// TIA Portal V20 export
// export: Created 2025-12-01T14:57:01.3679822Z, ExportSetting None, DisplayName Totally Integrated Automation Portal, DisplayVersion V20 Update 3, DisplayName TIA Portal Openness, DisplayVersion V20 Update 3, DisplayName TIA Portal Version Control Interface, DisplayVersion V20 Update 3, DisplayName STEP 7 Professional, DisplayVersion V20 Update 3, DisplayName STEP 7 Safety, DisplayVersion V20 Update 2, DisplayName WinCC Basic/Comfort/Advanced, DisplayVersion V20 Update 3, DisplayName WinCC Professional, DisplayVersion V20 Update 3, DisplayName WinCC Unified, DisplayVersion V20 Update 3
FUNCTION "FC457_TL_TR_E1E3_S2_Aus" : Void   // FC457, LAD
{ S7_Optimized_Access := 'FALSE' }
AUTHOR : TLigero
NAME : 20180125
VERSION : 3.2
// FECHA:    27/07/2014  AUTOR: G.Martin
// INSTALACION: Magyar Posta
// //////////////////////////////////
// // Registro Incidencias   ////////
// //////////////////////////////////
// FECHA:21/10/14   AUTOR MODIFICACION: N.Rodriguez
// DESCRIPCION: 
// Adaptación de la función al estandar actual
// ULTIMA MODIFICACION: iñaki Arrondo por problemas detectados en la instalacion (ALKAR)
// stored: AutoNumber false, SetENOAutomatically false
   VAR_INPUT
      Mesa : UInt;
      En_Tension : Bool;
      pHsMx_E1 : Bool;
      pHsMx_E3 : Bool;
      pHsMx_S2 : Bool;
      TP_E1_UP : Bool;
      TP_E1_Dw : Bool;
      TP_E3_UP : Bool;
      TP_E3_Dw : Bool;
      Termico_E1_Tx : Bool;
      Termico_S2_Tx : Bool;
      Avance_E1_Tx_Ok : Bool;
      Avance_E3_Tx_Ok : Bool;   // será el retroceso de E1
      Avance_S2_Tx_Ok : Bool;
      PosTR_E1 : Bool;
      PosTR_S2 : Bool;
      AVTF_Ent_M1 : Bool;
      AVTF_Ent_M3 : Bool;
      NXT_Avance : Bool;
      PTF_Mx_MSig : Bool;
      V_CNT_ApHsMx_S2 : UDInt;   // Valor del Contador de ausencia en S2
      V_CNT_ApHsMx_E1 : UDInt;   // Valor del Contador de ausencia en E1
      V_CNT_ApHsMx_E3 : UDInt;   // Valor del Contador de ausencia en S3
      V_Paro : UDInt;
      V_TOut_Tx_Mx : UDInt;
      V_TOut_TR : UDInt;
      V_RepartoColector : UDInt;
   END_VAR
   VAR_OUTPUT
      PTF_Ent_M1 : Bool;
      PTF_Ent_M3 : Bool;
      AVTF_Mx_MSig : Bool;
   END_VAR
   VAR_IN_OUT
      Mem_tmp_Paro : Bool;
      MemAuxFN_E1 : Bool;
      MemFN_pHsE1 : Bool;
      MemFP_pHsE1 : Bool;
      MemAuxFN_E3 : Bool;
      MemFN_pHsE3 : Bool;
      MemAuxFN_S2 : Bool;
      MemFN_pHsS2 : Bool;
   END_VAR
   VAR_TEMP
      OK_Ausencia_Entrada : Bool;
      OK_Ausencia_salida : Bool;
      ok_vaciado : Bool;
      Error_Atasco : Bool;
      Error_TOut_TR : Bool;
      TEMP_MA_TR_PosE1E3 : Bool;
      TEMP_MA_TR_PosS2 : Bool;
      ok_tension : Bool;
      v_ausencia_entrada : UDInt;
   END_VAR
   VAR_TEMP   // added for the SCL form of the ladder/FBD networks
      _w1 : Bool;
      _w2 : Bool;
      _w3 : Bool;
      _w4 : Bool;
      _w5 : Bool;
      _w6 : Bool;
   END_VAR
BEGIN

REGION Network 1: Marca General Error
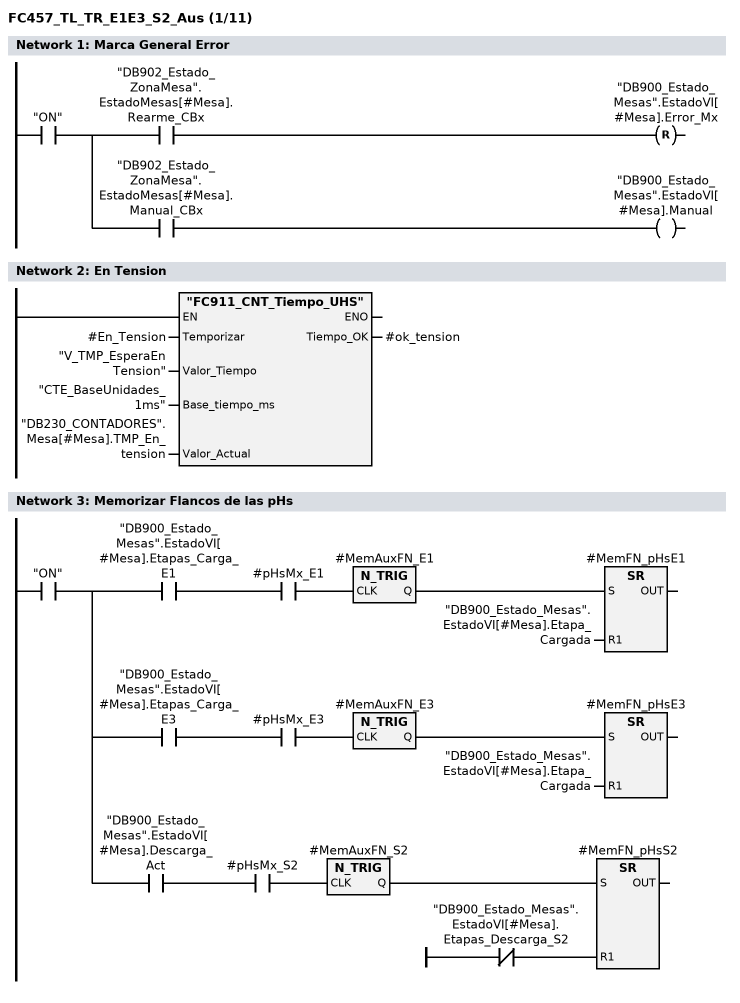
   RUNG wire#powerrail
      Contact( "ON" )
      wire#w1
      Contact( "DB902_Estado_ZonaMesa".EstadoMesas[#Mesa].Rearme_CBx )
      R_Coil( "DB900_Estado_Mesas".EstadoVI[#Mesa].Error_Mx )
   END_RUNG
   RUNG wire#w1
      Contact( "DB902_Estado_ZonaMesa".EstadoMesas[#Mesa].Manual_CBx )
      Coil( "DB900_Estado_Mesas".EstadoVI[#Mesa].Manual )
   END_RUNG
   // the same network as SCL:
   IF "ON" AND "DB902_Estado_ZonaMesa".EstadoMesas[#Mesa].Rearme_CBx THEN
       "DB900_Estado_Mesas".EstadoVI[#Mesa].Error_Mx := FALSE;
   END_IF;
   "DB900_Estado_Mesas".EstadoVI[#Mesa].Manual := "ON" AND "DB902_Estado_ZonaMesa".EstadoMesas[#Mesa].Manual_CBx;
END_REGION

REGION Network 2: En Tension
   RUNG wire#powerrail
      "FC911_CNT_Tiempo_UHS"(Temporizar := #En_Tension, Valor_Tiempo := "V_TMP_EsperaEnTension", Base_tiempo_ms := "CTE_BaseUnidades_1ms", Valor_Actual := "DB230_CONTADORES".Mesa[#Mesa].TMP_En_tension, Tiempo_OK => #ok_tension)
   END_RUNG
   // the same network as SCL:
   "FC911_CNT_Tiempo_UHS"(Temporizar := #En_Tension,
                          Valor_Tiempo := "V_TMP_EsperaEnTension",
                          Base_tiempo_ms := "CTE_BaseUnidades_1ms",
                          Valor_Actual := "DB230_CONTADORES".Mesa[#Mesa].TMP_En_tension,
                          Tiempo_OK => #ok_tension);
END_REGION

REGION Network 3: Memorizar Flancos de las pHs
   RUNG wire#powerrail
      Contact( "ON" )
      wire#w1
      Contact( "DB900_Estado_Mesas".EstadoVI[#Mesa].Etapas_Carga_E1 )
      Contact( #pHsMx_E1 )
      N_Trig( #MemAuxFN_E1 )
      S_SR(operand := #MemFN_pHsE1, r1 := "DB900_Estado_Mesas".EstadoVI[#Mesa].Etapa_Cargada)
   END_RUNG
   RUNG wire#w1
      Contact( "DB900_Estado_Mesas".EstadoVI[#Mesa].Etapas_Carga_E3 )
      Contact( #pHsMx_E3 )
      N_Trig( #MemAuxFN_E3 )
      S_SR(operand := #MemFN_pHsE3, r1 := "DB900_Estado_Mesas".EstadoVI[#Mesa].Etapa_Cargada)
   END_RUNG
   RUNG wire#w1
      Contact( "DB900_Estado_Mesas".EstadoVI[#Mesa].Descarga_Act )
      Contact( #pHsMx_S2 )
      N_Trig( #MemAuxFN_S2 )
      S_SR(operand := #MemFN_pHsS2, r1 := wire#w2)
   END_RUNG
   RUNG wire#powerrail
      I_Contact( "DB900_Estado_Mesas".EstadoVI[#Mesa].Etapas_Descarga_S2 )
   END_RUNG wire#w2
   // the same network as SCL:
   #_w1 := "ON" AND "DB900_Estado_Mesas".EstadoVI[#Mesa].Etapas_Carga_E1 AND #pHsMx_E1;
   #_w2 := NOT #_w1 AND #MemAuxFN_E1;   // falling edge
   #MemAuxFN_E1 := #_w1;
   IF #_w2 THEN
       #MemFN_pHsE1 := TRUE;   // SR flip-flop
   END_IF;
   IF "DB900_Estado_Mesas".EstadoVI[#Mesa].Etapa_Cargada THEN #MemFN_pHsE1 := FALSE; END_IF;
   #_w3 := "ON" AND "DB900_Estado_Mesas".EstadoVI[#Mesa].Etapas_Carga_E3 AND #pHsMx_E3;
   #_w4 := NOT #_w3 AND #MemAuxFN_E3;   // falling edge
   #MemAuxFN_E3 := #_w3;
   IF #_w4 THEN
       #MemFN_pHsE3 := TRUE;   // SR flip-flop
   END_IF;
   IF "DB900_Estado_Mesas".EstadoVI[#Mesa].Etapa_Cargada THEN #MemFN_pHsE3 := FALSE; END_IF;
   #_w5 := "ON" AND "DB900_Estado_Mesas".EstadoVI[#Mesa].Descarga_Act AND #pHsMx_S2;
   #_w6 := NOT #_w5 AND #MemAuxFN_S2;   // falling edge
   #MemAuxFN_S2 := #_w5;
   IF #_w6 THEN
       #MemFN_pHsS2 := TRUE;   // SR flip-flop
   END_IF;
   IF NOT "DB900_Estado_Mesas".EstadoVI[#Mesa].Etapas_Descarga_S2 THEN #MemFN_pHsS2 := FALSE; END_IF;
END_REGION

REGION Network 4: contador vaciado
   // Contador ausencia
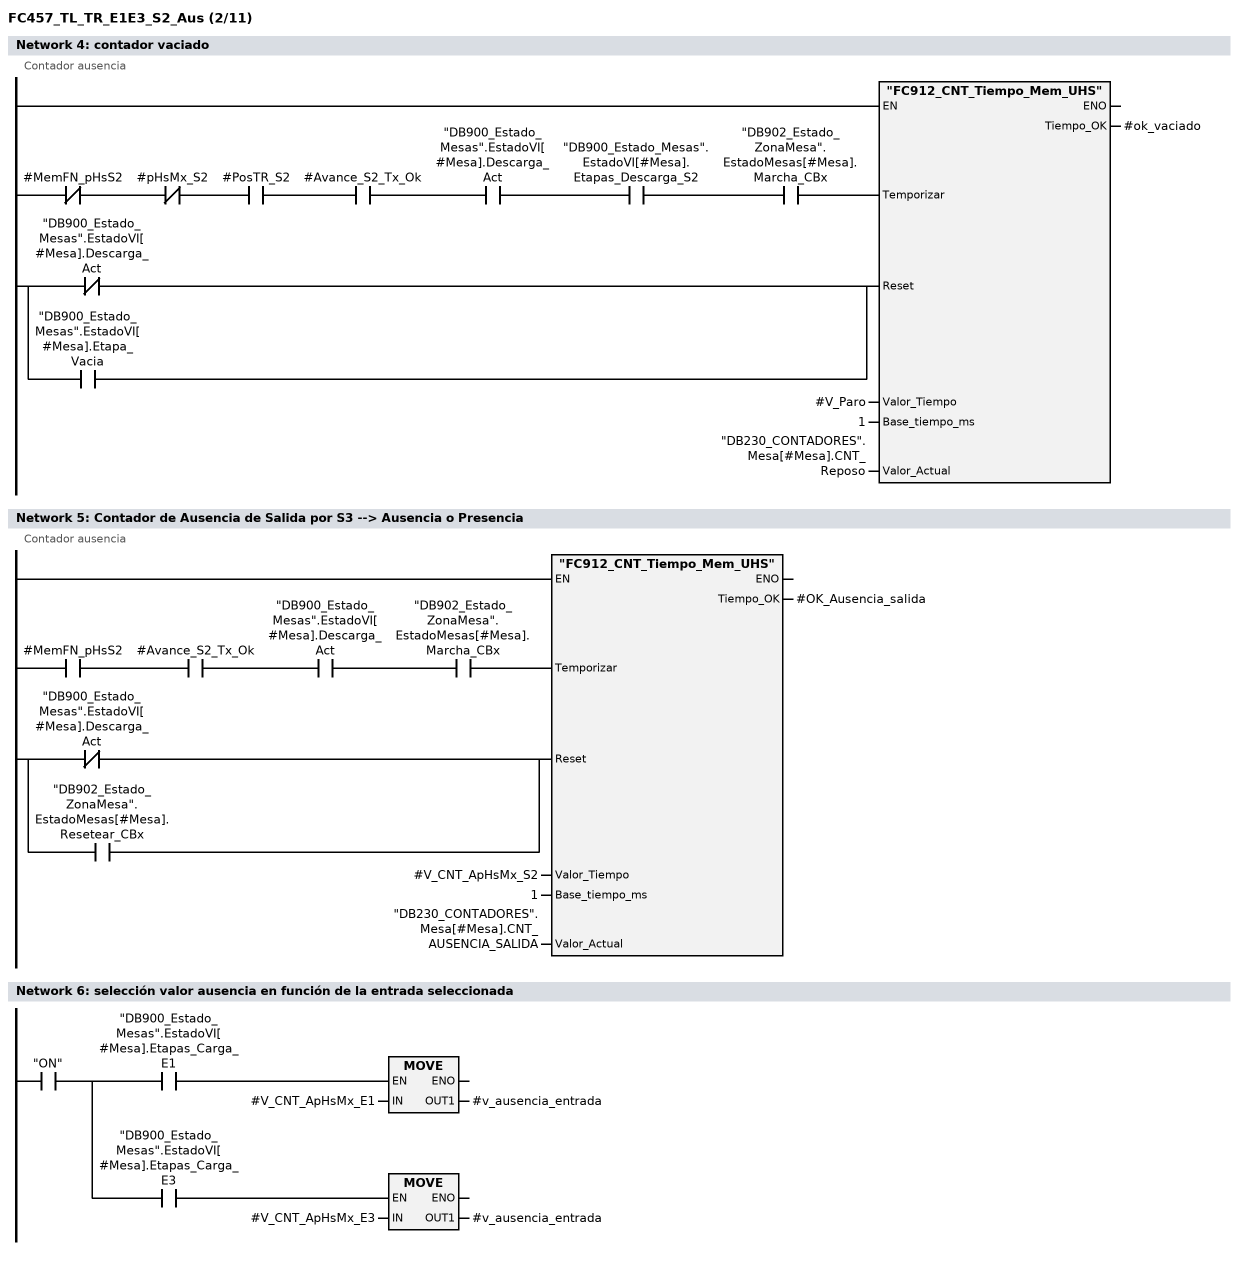
   RUNG wire#powerrail
      "FC912_CNT_Tiempo_Mem_UHS"(Temporizar := wire#w1, Reset := wire#w2, Valor_Tiempo := #V_Paro, Base_tiempo_ms := 1, Valor_Actual := "DB230_CONTADORES".Mesa[#Mesa].CNT_Reposo, Tiempo_OK => #ok_vaciado)
   END_RUNG
   RUNG wire#powerrail
      I_Contact( #MemFN_pHsS2 )
      I_Contact( #pHsMx_S2 )
      Contact( #PosTR_S2 )
      Contact( #Avance_S2_Tx_Ok )
      Contact( "DB900_Estado_Mesas".EstadoVI[#Mesa].Descarga_Act )
      Contact( "DB900_Estado_Mesas".EstadoVI[#Mesa].Etapas_Descarga_S2 )
      Contact( "DB902_Estado_ZonaMesa".EstadoMesas[#Mesa].Marcha_CBx )
   END_RUNG wire#w1
   RUNG wire#powerrail
      I_Contact( "DB900_Estado_Mesas".EstadoVI[#Mesa].Descarga_Act )
   END_RUNG wire#w2
   RUNG wire#powerrail
      Contact( "DB900_Estado_Mesas".EstadoVI[#Mesa].Etapa_Vacia )
   END_RUNG wire#w2
   // the same network as SCL:
   "FC912_CNT_Tiempo_Mem_UHS"(Temporizar := NOT #MemFN_pHsS2 AND NOT #pHsMx_S2 AND #PosTR_S2 AND #Avance_S2_Tx_Ok AND "DB900_Estado_Mesas".EstadoVI[#Mesa].Descarga_Act AND "DB900_Estado_Mesas".EstadoVI[#Mesa].Etapas_Descarga_S2 AND "DB902_Estado_ZonaMesa".EstadoMesas[#Mesa].Marcha_CBx,
                           Reset := NOT "DB900_Estado_Mesas".EstadoVI[#Mesa].Descarga_Act OR "DB900_Estado_Mesas".EstadoVI[#Mesa].Etapa_Vacia,
                           Valor_Tiempo := #V_Paro,
                           Base_tiempo_ms := 1,
                           Valor_Actual := "DB230_CONTADORES".Mesa[#Mesa].CNT_Reposo,
                           Tiempo_OK => #ok_vaciado);
END_REGION

REGION Network 5: Contador de Ausencia de Salida por S3 --> Ausencia o Presencia
   // Contador ausencia
   RUNG wire#powerrail
      "FC912_CNT_Tiempo_Mem_UHS"(Temporizar := wire#w1, Reset := wire#w2, Valor_Tiempo := #V_CNT_ApHsMx_S2, Base_tiempo_ms := 1, Valor_Actual := "DB230_CONTADORES".Mesa[#Mesa].CNT_AUSENCIA_SALIDA, Tiempo_OK => #OK_Ausencia_salida)
   END_RUNG
   RUNG wire#powerrail
      Contact( #MemFN_pHsS2 )
      Contact( #Avance_S2_Tx_Ok )
      Contact( "DB900_Estado_Mesas".EstadoVI[#Mesa].Descarga_Act )
      Contact( "DB902_Estado_ZonaMesa".EstadoMesas[#Mesa].Marcha_CBx )
   END_RUNG wire#w1
   RUNG wire#powerrail
      I_Contact( "DB900_Estado_Mesas".EstadoVI[#Mesa].Descarga_Act )
   END_RUNG wire#w2
   RUNG wire#powerrail
      Contact( "DB902_Estado_ZonaMesa".EstadoMesas[#Mesa].Resetear_CBx )
   END_RUNG wire#w2
   // the same network as SCL:
   "FC912_CNT_Tiempo_Mem_UHS"(Temporizar := #MemFN_pHsS2 AND #Avance_S2_Tx_Ok AND "DB900_Estado_Mesas".EstadoVI[#Mesa].Descarga_Act AND "DB902_Estado_ZonaMesa".EstadoMesas[#Mesa].Marcha_CBx,
                           Reset := NOT "DB900_Estado_Mesas".EstadoVI[#Mesa].Descarga_Act OR "DB902_Estado_ZonaMesa".EstadoMesas[#Mesa].Resetear_CBx,
                           Valor_Tiempo := #V_CNT_ApHsMx_S2,
                           Base_tiempo_ms := 1,
                           Valor_Actual := "DB230_CONTADORES".Mesa[#Mesa].CNT_AUSENCIA_SALIDA,
                           Tiempo_OK => #OK_Ausencia_salida);
END_REGION

REGION Network 6: selección valor ausencia en función de la entrada seleccionada
   RUNG wire#powerrail
      Contact( "ON" )
      wire#w1
      Contact( "DB900_Estado_Mesas".EstadoVI[#Mesa].Etapas_Carga_E1 )
      Move(in := #V_CNT_ApHsMx_E1, out1 => #v_ausencia_entrada)
   END_RUNG
   RUNG wire#w1
      Contact( "DB900_Estado_Mesas".EstadoVI[#Mesa].Etapas_Carga_E3 )
      Move(in := #V_CNT_ApHsMx_E3, out1 => #v_ausencia_entrada)
   END_RUNG
   // the same network as SCL:
   IF "ON" AND "DB900_Estado_Mesas".EstadoVI[#Mesa].Etapas_Carga_E1 THEN
       #v_ausencia_entrada := #V_CNT_ApHsMx_E1;
   END_IF;
   IF "ON" AND "DB900_Estado_Mesas".EstadoVI[#Mesa].Etapas_Carga_E3 THEN
       #v_ausencia_entrada := #V_CNT_ApHsMx_E3;
   END_IF;
END_REGION

REGION Network 7: Contador de Ausencia de Entrada
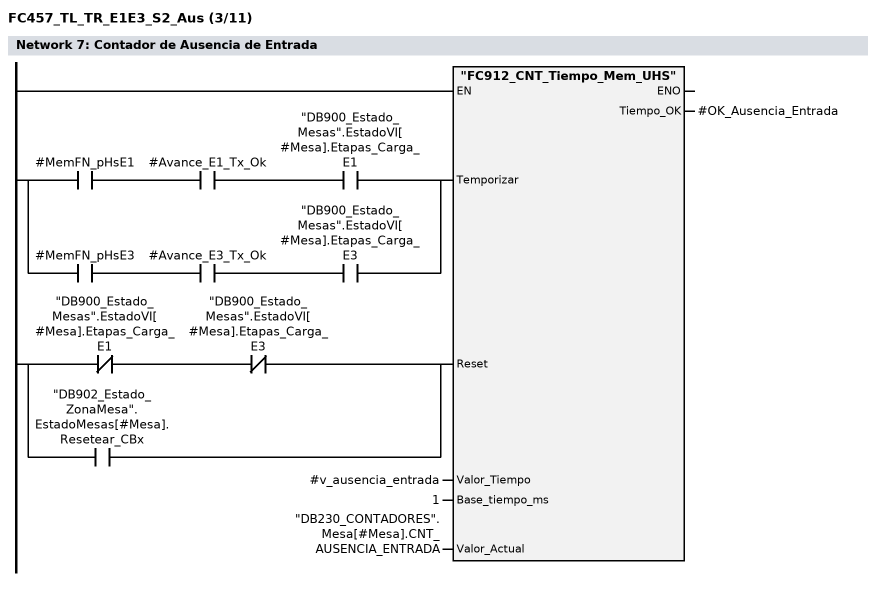
   RUNG wire#powerrail
      "FC912_CNT_Tiempo_Mem_UHS"(Temporizar := wire#w1, Reset := wire#w2, Valor_Tiempo := #v_ausencia_entrada, Base_tiempo_ms := 1, Valor_Actual := "DB230_CONTADORES".Mesa[#Mesa].CNT_AUSENCIA_ENTRADA, Tiempo_OK => #OK_Ausencia_Entrada)
   END_RUNG
   RUNG wire#powerrail
      Contact( #MemFN_pHsE1 )
      Contact( #Avance_E1_Tx_Ok )
      Contact( "DB900_Estado_Mesas".EstadoVI[#Mesa].Etapas_Carga_E1 )
   END_RUNG wire#w1
   RUNG wire#powerrail
      Contact( #MemFN_pHsE3 )
      Contact( #Avance_E3_Tx_Ok )
      Contact( "DB900_Estado_Mesas".EstadoVI[#Mesa].Etapas_Carga_E3 )
   END_RUNG wire#w1
   RUNG wire#powerrail
      I_Contact( "DB900_Estado_Mesas".EstadoVI[#Mesa].Etapas_Carga_E1 )
      I_Contact( "DB900_Estado_Mesas".EstadoVI[#Mesa].Etapas_Carga_E3 )
   END_RUNG wire#w2
   RUNG wire#powerrail
      Contact( "DB902_Estado_ZonaMesa".EstadoMesas[#Mesa].Resetear_CBx )
   END_RUNG wire#w2
   // the same network as SCL:
   "FC912_CNT_Tiempo_Mem_UHS"(Temporizar := (#MemFN_pHsE1 AND #Avance_E1_Tx_Ok AND "DB900_Estado_Mesas".EstadoVI[#Mesa].Etapas_Carga_E1) OR (#MemFN_pHsE3 AND #Avance_E3_Tx_Ok AND "DB900_Estado_Mesas".EstadoVI[#Mesa].Etapas_Carga_E3),
                           Reset := (NOT "DB900_Estado_Mesas".EstadoVI[#Mesa].Etapas_Carga_E1 AND NOT "DB900_Estado_Mesas".EstadoVI[#Mesa].Etapas_Carga_E3) OR "DB902_Estado_ZonaMesa".EstadoMesas[#Mesa].Resetear_CBx,
                           Valor_Tiempo := #v_ausencia_entrada,
                           Base_tiempo_ms := 1,
                           Valor_Actual := "DB230_CONTADORES".Mesa[#Mesa].CNT_AUSENCIA_ENTRADA,
                           Tiempo_OK => #OK_Ausencia_Entrada);
END_REGION

REGION Network 8: Temporizador de PARO
   // Modif Dani: El contador se activa además de con MA_avance_Tx, con el 
   // MA_Avance_TR, pq sino, no se resetean las variables de Mem_Act_E1, E2 tras un 
   // reset
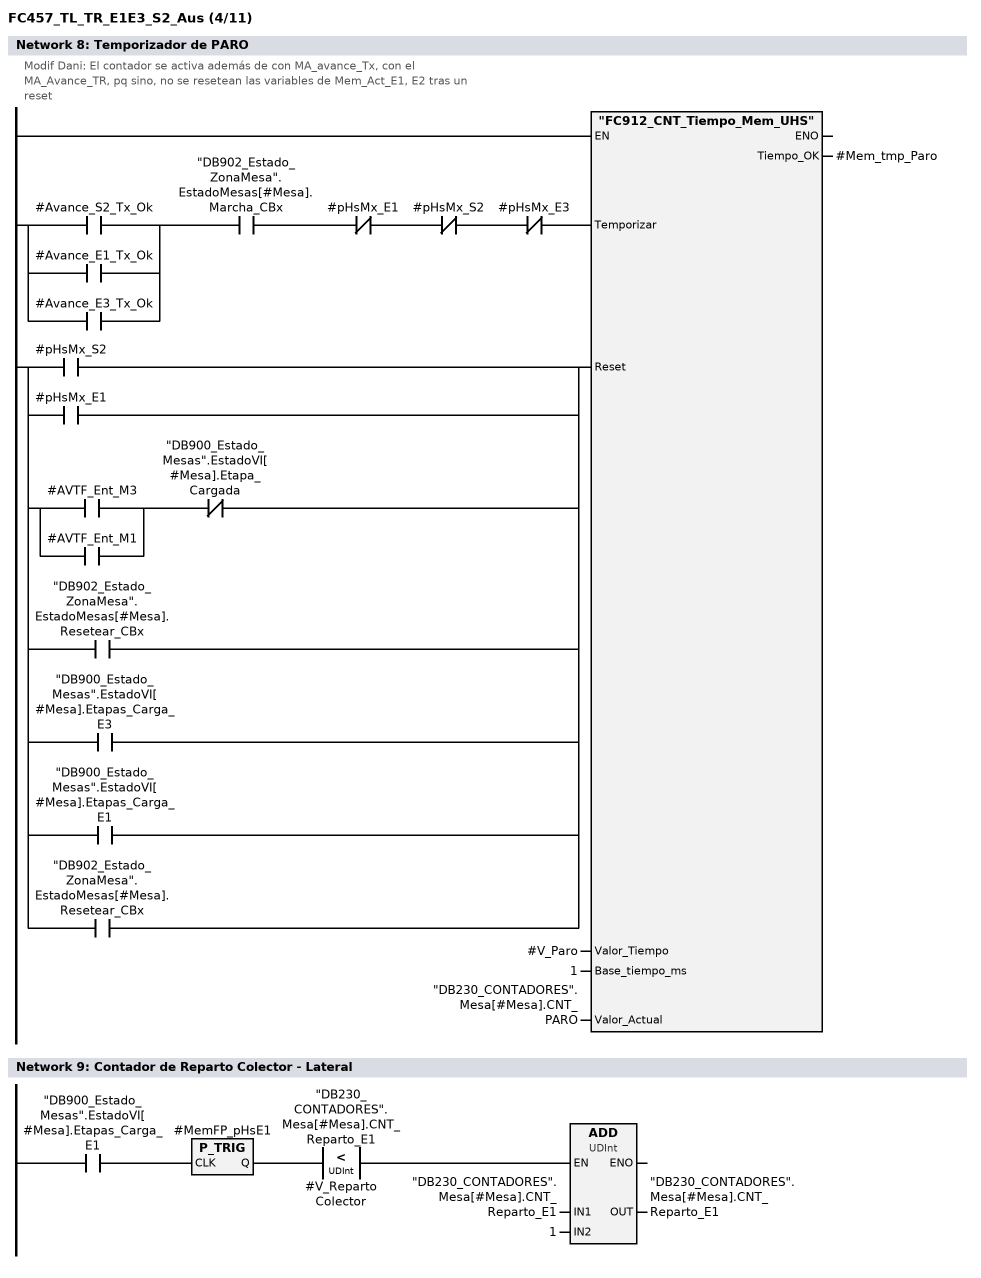
   RUNG wire#powerrail
      "FC912_CNT_Tiempo_Mem_UHS"(Temporizar := wire#w2, Reset := wire#w4, Valor_Tiempo := #V_Paro, Base_tiempo_ms := 1, Valor_Actual := "DB230_CONTADORES".Mesa[#Mesa].CNT_PARO, Tiempo_OK => #Mem_tmp_Paro)
   END_RUNG
   RUNG wire#powerrail
      Contact( #Avance_S2_Tx_Ok )
      wire#w1
      Contact( "DB902_Estado_ZonaMesa".EstadoMesas[#Mesa].Marcha_CBx )
      I_Contact( #pHsMx_E1 )
      I_Contact( #pHsMx_S2 )
      I_Contact( #pHsMx_E3 )
   END_RUNG wire#w2
   RUNG wire#powerrail
      Contact( #Avance_E1_Tx_Ok )
   END_RUNG wire#w1
   RUNG wire#powerrail
      Contact( #Avance_E3_Tx_Ok )
   END_RUNG wire#w1
   RUNG wire#powerrail
      Contact( #pHsMx_S2 )
   END_RUNG wire#w4
   RUNG wire#powerrail
      Contact( #pHsMx_E1 )
   END_RUNG wire#w4
   RUNG wire#powerrail
      Contact( #AVTF_Ent_M3 )
      wire#w3
      I_Contact( "DB900_Estado_Mesas".EstadoVI[#Mesa].Etapa_Cargada )
   END_RUNG wire#w4
   RUNG wire#powerrail
      Contact( #AVTF_Ent_M1 )
   END_RUNG wire#w3
   RUNG wire#powerrail
      Contact( "DB902_Estado_ZonaMesa".EstadoMesas[#Mesa].Resetear_CBx )
   END_RUNG wire#w4
   RUNG wire#powerrail
      Contact( "DB900_Estado_Mesas".EstadoVI[#Mesa].Etapas_Carga_E3 )
   END_RUNG wire#w4
   RUNG wire#powerrail
      Contact( "DB900_Estado_Mesas".EstadoVI[#Mesa].Etapas_Carga_E1 )
   END_RUNG wire#w4
   RUNG wire#powerrail
      Contact( "DB902_Estado_ZonaMesa".EstadoMesas[#Mesa].Resetear_CBx )
   END_RUNG wire#w4
   // the same network as SCL:
   "FC912_CNT_Tiempo_Mem_UHS"(Temporizar := (#Avance_S2_Tx_Ok OR #Avance_E1_Tx_Ok OR #Avance_E3_Tx_Ok) AND "DB902_Estado_ZonaMesa".EstadoMesas[#Mesa].Marcha_CBx AND NOT #pHsMx_E1 AND NOT #pHsMx_S2 AND NOT #pHsMx_E3,
                           Reset := #pHsMx_S2 OR #pHsMx_E1 OR ((#AVTF_Ent_M3 OR #AVTF_Ent_M1) AND NOT "DB900_Estado_Mesas".EstadoVI[#Mesa].Etapa_Cargada) OR "DB902_Estado_ZonaMesa".EstadoMesas[#Mesa].Resetear_CBx OR "DB900_Estado_Mesas".EstadoVI[#Mesa].Etapas_Carga_E3 OR "DB900_Estado_Mesas".EstadoVI[#Mesa].Etapas_Carga_E1 OR "DB902_Estado_ZonaMesa".EstadoMesas[#Mesa].Resetear_CBx,
                           Valor_Tiempo := #V_Paro,
                           Base_tiempo_ms := 1,
                           Valor_Actual := "DB230_CONTADORES".Mesa[#Mesa].CNT_PARO,
                           Tiempo_OK => #Mem_tmp_Paro);
END_REGION

REGION Network 9: Contador de Reparto Colector - Lateral
   RUNG wire#powerrail
      Contact( "DB900_Estado_Mesas".EstadoVI[#Mesa].Etapas_Carga_E1 )
      P_Trig( #MemFP_pHsE1 )
      { S7_Templates := "SrcType := UDInt" } LT_Contact(in1 := "DB230_CONTADORES".Mesa[#Mesa].CNT_Reparto_E1, in2 := #V_RepartoColector)
      { S7_Templates := "SrcType := UDInt"; S7_GenerateENO := "TRUE" } Add(in1 := "DB230_CONTADORES".Mesa[#Mesa].CNT_Reparto_E1, in2 := 1, out => "DB230_CONTADORES".Mesa[#Mesa].CNT_Reparto_E1)
   END_RUNG
   // the same network as SCL:
   #_w1 := "DB900_Estado_Mesas".EstadoVI[#Mesa].Etapas_Carga_E1 AND NOT #MemFP_pHsE1;   // rising edge
   #MemFP_pHsE1 := "DB900_Estado_Mesas".EstadoVI[#Mesa].Etapas_Carga_E1;
   IF #_w1 AND ("DB230_CONTADORES".Mesa[#Mesa].CNT_Reparto_E1 < #V_RepartoColector) THEN
       "DB230_CONTADORES".Mesa[#Mesa].CNT_Reparto_E1 := "DB230_CONTADORES".Mesa[#Mesa].CNT_Reparto_E1 + 1;
   END_IF;
END_REGION

REGION Network 10
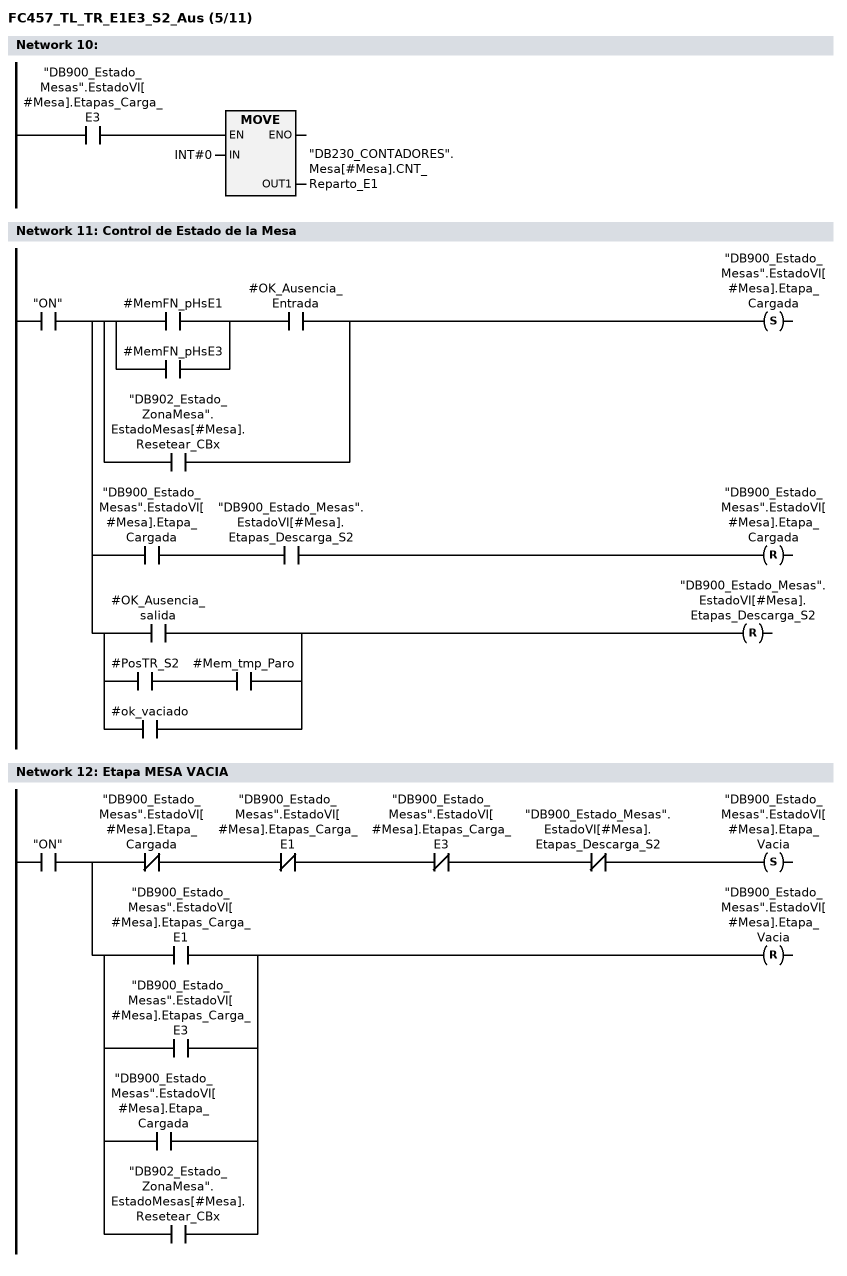
   RUNG wire#powerrail
      Contact( "DB900_Estado_Mesas".EstadoVI[#Mesa].Etapas_Carga_E3 )
      { S7_GenerateENO := "TRUE" } Move(in := INT#0, out1 => "DB230_CONTADORES".Mesa[#Mesa].CNT_Reparto_E1)
   END_RUNG
   // the same network as SCL:
   IF "DB900_Estado_Mesas".EstadoVI[#Mesa].Etapas_Carga_E3 THEN
       "DB230_CONTADORES".Mesa[#Mesa].CNT_Reparto_E1 := INT#0;
   END_IF;
END_REGION

REGION Network 11: Control de Estado de la Mesa
   RUNG wire#powerrail
      Contact( "ON" )
      wire#w1
      Contact( #MemFN_pHsE1 )
      wire#w2
      Contact( #OK_Ausencia_Entrada )
      wire#w3
      S_Coil( "DB900_Estado_Mesas".EstadoVI[#Mesa].Etapa_Cargada )
   END_RUNG
   RUNG wire#w1
      Contact( #MemFN_pHsE3 )
   END_RUNG wire#w2
   RUNG wire#w1
      Contact( "DB902_Estado_ZonaMesa".EstadoMesas[#Mesa].Resetear_CBx )
   END_RUNG wire#w3
   RUNG wire#w1
      Contact( "DB900_Estado_Mesas".EstadoVI[#Mesa].Etapa_Cargada )
      Contact( "DB900_Estado_Mesas".EstadoVI[#Mesa].Etapas_Descarga_S2 )
      R_Coil( "DB900_Estado_Mesas".EstadoVI[#Mesa].Etapa_Cargada )
   END_RUNG
   RUNG wire#w1
      Contact( #OK_Ausencia_salida )
      wire#w4
      R_Coil( "DB900_Estado_Mesas".EstadoVI[#Mesa].Etapas_Descarga_S2 )
   END_RUNG
   RUNG wire#w1
      Contact( #PosTR_S2 )
      Contact( #Mem_tmp_Paro )
   END_RUNG wire#w4
   RUNG wire#w1
      Contact( #ok_vaciado )
   END_RUNG wire#w4
   // the same network as SCL:
   IF "ON" AND (((#MemFN_pHsE1 OR #MemFN_pHsE3) AND #OK_Ausencia_Entrada) OR "DB902_Estado_ZonaMesa".EstadoMesas[#Mesa].Resetear_CBx) THEN
       "DB900_Estado_Mesas".EstadoVI[#Mesa].Etapa_Cargada := TRUE;
   END_IF;
   IF "ON" AND "DB900_Estado_Mesas".EstadoVI[#Mesa].Etapa_Cargada AND "DB900_Estado_Mesas".EstadoVI[#Mesa].Etapas_Descarga_S2 THEN
       "DB900_Estado_Mesas".EstadoVI[#Mesa].Etapa_Cargada := FALSE;
   END_IF;
   IF "ON" AND (#OK_Ausencia_salida OR (#PosTR_S2 AND #Mem_tmp_Paro) OR #ok_vaciado) THEN
       "DB900_Estado_Mesas".EstadoVI[#Mesa].Etapas_Descarga_S2 := FALSE;
   END_IF;
END_REGION

REGION Network 12: Etapa MESA VACIA
   RUNG wire#powerrail
      Contact( "ON" )
      wire#w1
      I_Contact( "DB900_Estado_Mesas".EstadoVI[#Mesa].Etapa_Cargada )
      I_Contact( "DB900_Estado_Mesas".EstadoVI[#Mesa].Etapas_Carga_E1 )
      I_Contact( "DB900_Estado_Mesas".EstadoVI[#Mesa].Etapas_Carga_E3 )
      I_Contact( "DB900_Estado_Mesas".EstadoVI[#Mesa].Etapas_Descarga_S2 )
      S_Coil( "DB900_Estado_Mesas".EstadoVI[#Mesa].Etapa_Vacia )
   END_RUNG
   RUNG wire#w1
      Contact( "DB900_Estado_Mesas".EstadoVI[#Mesa].Etapas_Carga_E1 )
      wire#w2
      R_Coil( "DB900_Estado_Mesas".EstadoVI[#Mesa].Etapa_Vacia )
   END_RUNG
   RUNG wire#w1
      Contact( "DB900_Estado_Mesas".EstadoVI[#Mesa].Etapas_Carga_E3 )
   END_RUNG wire#w2
   RUNG wire#w1
      Contact( "DB900_Estado_Mesas".EstadoVI[#Mesa].Etapa_Cargada )
   END_RUNG wire#w2
   RUNG wire#w1
      Contact( "DB902_Estado_ZonaMesa".EstadoMesas[#Mesa].Resetear_CBx )
   END_RUNG wire#w2
   // the same network as SCL:
   IF "ON" AND NOT "DB900_Estado_Mesas".EstadoVI[#Mesa].Etapa_Cargada AND NOT "DB900_Estado_Mesas".EstadoVI[#Mesa].Etapas_Carga_E1 AND NOT "DB900_Estado_Mesas".EstadoVI[#Mesa].Etapas_Carga_E3 AND NOT "DB900_Estado_Mesas".EstadoVI[#Mesa].Etapas_Descarga_S2 THEN
       "DB900_Estado_Mesas".EstadoVI[#Mesa].Etapa_Vacia := TRUE;
   END_IF;
   IF "ON" AND ("DB900_Estado_Mesas".EstadoVI[#Mesa].Etapas_Carga_E1 OR "DB900_Estado_Mesas".EstadoVI[#Mesa].Etapas_Carga_E3 OR "DB900_Estado_Mesas".EstadoVI[#Mesa].Etapa_Cargada OR "DB902_Estado_ZonaMesa".EstadoMesas[#Mesa].Resetear_CBx) THEN
       "DB900_Estado_Mesas".EstadoVI[#Mesa].Etapa_Vacia := FALSE;
   END_IF;
END_REGION

REGION Network 13
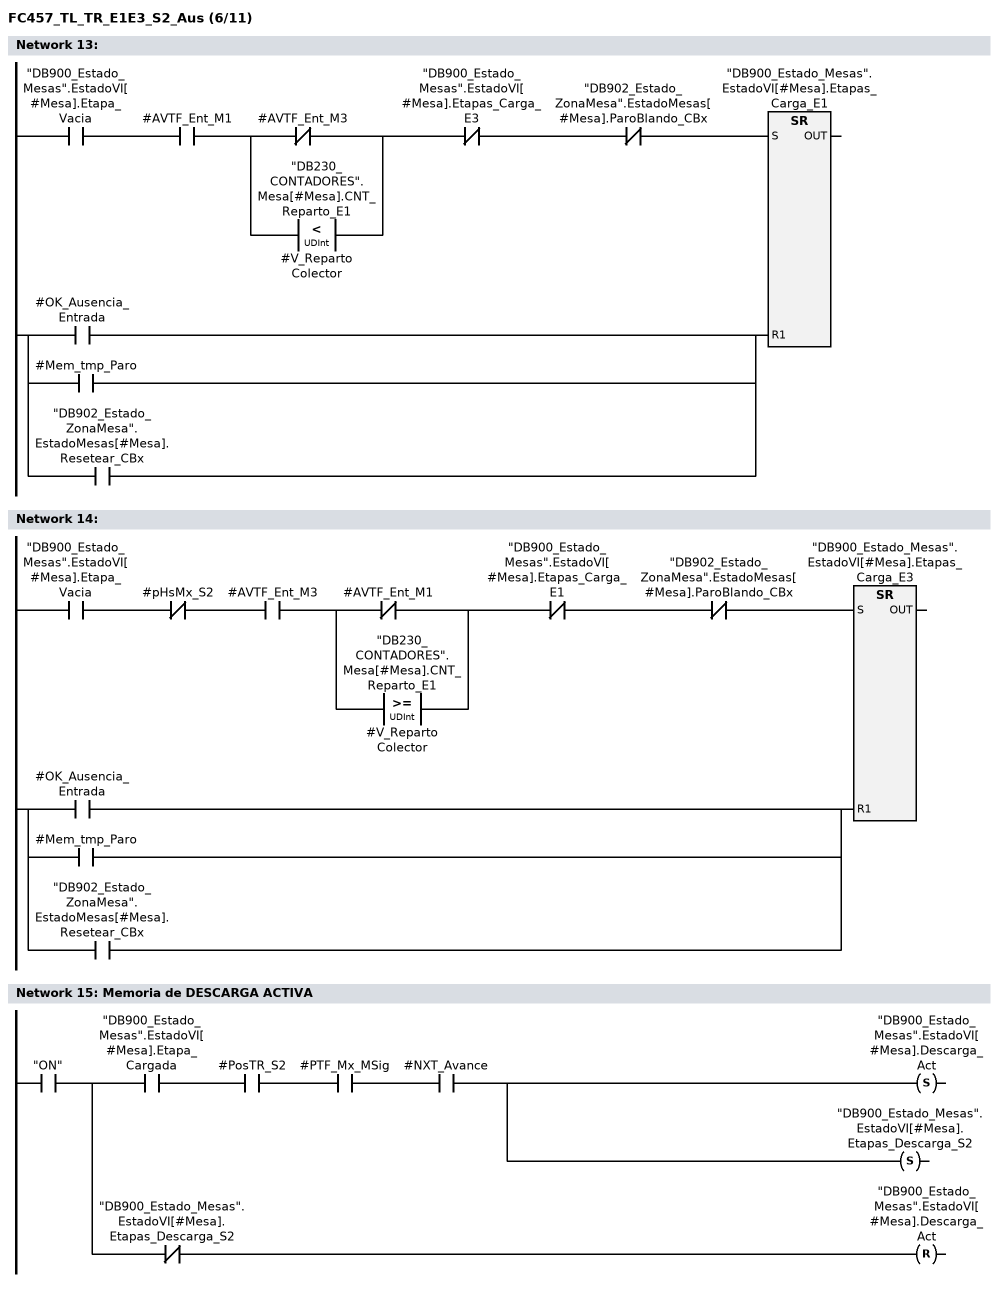
   RUNG wire#powerrail
      Contact( "DB900_Estado_Mesas".EstadoVI[#Mesa].Etapa_Vacia )
      Contact( #AVTF_Ent_M1 )
      wire#w1
      I_Contact( #AVTF_Ent_M3 )
      wire#w2
      I_Contact( "DB900_Estado_Mesas".EstadoVI[#Mesa].Etapas_Carga_E3 )
      I_Contact( "DB902_Estado_ZonaMesa".EstadoMesas[#Mesa].ParoBlando_CBx )
      S_SR(operand := "DB900_Estado_Mesas".EstadoVI[#Mesa].Etapas_Carga_E1, r1 := wire#w3)
   END_RUNG
   RUNG wire#w1
      { S7_Templates := "SrcType := UDInt" } LT_Contact(in1 := "DB230_CONTADORES".Mesa[#Mesa].CNT_Reparto_E1, in2 := #V_RepartoColector)
   END_RUNG wire#w2
   RUNG wire#powerrail
      Contact( #OK_Ausencia_Entrada )
   END_RUNG wire#w3
   RUNG wire#powerrail
      Contact( #Mem_tmp_Paro )
   END_RUNG wire#w3
   RUNG wire#powerrail
      Contact( "DB902_Estado_ZonaMesa".EstadoMesas[#Mesa].Resetear_CBx )
   END_RUNG wire#w3
   // the same network as SCL:
   #_w1 := #OK_Ausencia_Entrada OR #Mem_tmp_Paro OR "DB902_Estado_ZonaMesa".EstadoMesas[#Mesa].Resetear_CBx;
   IF "DB900_Estado_Mesas".EstadoVI[#Mesa].Etapa_Vacia AND #AVTF_Ent_M1 AND (NOT #AVTF_Ent_M3 OR ("DB230_CONTADORES".Mesa[#Mesa].CNT_Reparto_E1 < #V_RepartoColector)) AND NOT "DB900_Estado_Mesas".EstadoVI[#Mesa].Etapas_Carga_E3 AND NOT "DB902_Estado_ZonaMesa".EstadoMesas[#Mesa].ParoBlando_CBx THEN
       "DB900_Estado_Mesas".EstadoVI[#Mesa].Etapas_Carga_E1 := TRUE;   // SR flip-flop
   END_IF;
   IF #_w1 THEN "DB900_Estado_Mesas".EstadoVI[#Mesa].Etapas_Carga_E1 := FALSE; END_IF;
END_REGION

REGION Network 14
   RUNG wire#powerrail
      Contact( "DB900_Estado_Mesas".EstadoVI[#Mesa].Etapa_Vacia )
      I_Contact( #pHsMx_S2 )
      Contact( #AVTF_Ent_M3 )
      wire#w1
      I_Contact( #AVTF_Ent_M1 )
      wire#w2
      I_Contact( "DB900_Estado_Mesas".EstadoVI[#Mesa].Etapas_Carga_E1 )
      I_Contact( "DB902_Estado_ZonaMesa".EstadoMesas[#Mesa].ParoBlando_CBx )
      S_SR(operand := "DB900_Estado_Mesas".EstadoVI[#Mesa].Etapas_Carga_E3, r1 := wire#w3)
   END_RUNG
   RUNG wire#w1
      { S7_Templates := "SrcType := UDInt" } GE_Contact(in1 := "DB230_CONTADORES".Mesa[#Mesa].CNT_Reparto_E1, in2 := #V_RepartoColector)
   END_RUNG wire#w2
   RUNG wire#powerrail
      Contact( #OK_Ausencia_Entrada )
   END_RUNG wire#w3
   RUNG wire#powerrail
      Contact( #Mem_tmp_Paro )
   END_RUNG wire#w3
   RUNG wire#powerrail
      Contact( "DB902_Estado_ZonaMesa".EstadoMesas[#Mesa].Resetear_CBx )
   END_RUNG wire#w3
   // the same network as SCL:
   #_w1 := #OK_Ausencia_Entrada OR #Mem_tmp_Paro OR "DB902_Estado_ZonaMesa".EstadoMesas[#Mesa].Resetear_CBx;
   IF "DB900_Estado_Mesas".EstadoVI[#Mesa].Etapa_Vacia AND NOT #pHsMx_S2 AND #AVTF_Ent_M3 AND (NOT #AVTF_Ent_M1 OR ("DB230_CONTADORES".Mesa[#Mesa].CNT_Reparto_E1 >= #V_RepartoColector)) AND NOT "DB900_Estado_Mesas".EstadoVI[#Mesa].Etapas_Carga_E1 AND NOT "DB902_Estado_ZonaMesa".EstadoMesas[#Mesa].ParoBlando_CBx THEN
       "DB900_Estado_Mesas".EstadoVI[#Mesa].Etapas_Carga_E3 := TRUE;   // SR flip-flop
   END_IF;
   IF #_w1 THEN "DB900_Estado_Mesas".EstadoVI[#Mesa].Etapas_Carga_E3 := FALSE; END_IF;
END_REGION

REGION Network 15: Memoria de DESCARGA ACTIVA
   RUNG wire#powerrail
      Contact( "ON" )
      wire#w1
      Contact( "DB900_Estado_Mesas".EstadoVI[#Mesa].Etapa_Cargada )
      Contact( #PosTR_S2 )
      Contact( #PTF_Mx_MSig )
      Contact( #NXT_Avance )
      wire#w2
      S_Coil( "DB900_Estado_Mesas".EstadoVI[#Mesa].Descarga_Act )
   END_RUNG
   RUNG wire#w2
      S_Coil( "DB900_Estado_Mesas".EstadoVI[#Mesa].Etapas_Descarga_S2 )
   END_RUNG
   RUNG wire#w1
      I_Contact( "DB900_Estado_Mesas".EstadoVI[#Mesa].Etapas_Descarga_S2 )
      R_Coil( "DB900_Estado_Mesas".EstadoVI[#Mesa].Descarga_Act )
   END_RUNG
   // the same network as SCL:
   #_w1 := "ON" AND "DB900_Estado_Mesas".EstadoVI[#Mesa].Etapa_Cargada AND #PosTR_S2 AND #PTF_Mx_MSig AND #NXT_Avance;
   IF #_w1 THEN
       "DB900_Estado_Mesas".EstadoVI[#Mesa].Descarga_Act := TRUE;
       "DB900_Estado_Mesas".EstadoVI[#Mesa].Etapas_Descarga_S2 := TRUE;
   END_IF;
   IF "ON" AND NOT "DB900_Estado_Mesas".EstadoVI[#Mesa].Etapas_Descarga_S2 THEN
       "DB900_Estado_Mesas".EstadoVI[#Mesa].Descarga_Act := FALSE;
   END_IF;
END_REGION

REGION Network 16: Salidas Auxiliares
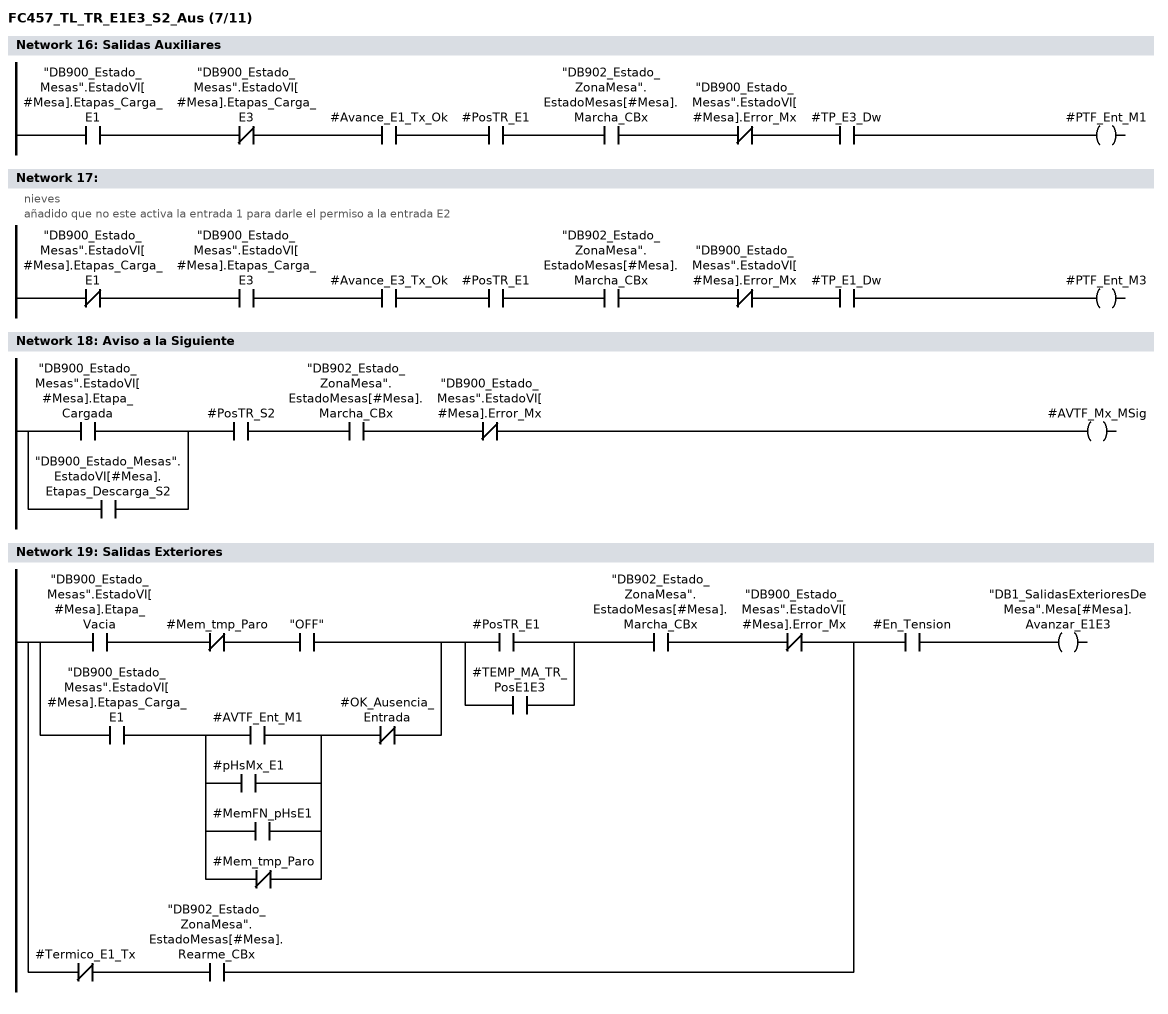
   RUNG wire#powerrail
      Contact( "DB900_Estado_Mesas".EstadoVI[#Mesa].Etapas_Carga_E1 )
      I_Contact( "DB900_Estado_Mesas".EstadoVI[#Mesa].Etapas_Carga_E3 )
      Contact( #Avance_E1_Tx_Ok )
      Contact( #PosTR_E1 )
      Contact( "DB902_Estado_ZonaMesa".EstadoMesas[#Mesa].Marcha_CBx )
      I_Contact( "DB900_Estado_Mesas".EstadoVI[#Mesa].Error_Mx )
      Contact( #TP_E3_Dw )
      Coil( #PTF_Ent_M1 )
   END_RUNG
   // the same network as SCL:
   #PTF_Ent_M1 := "DB900_Estado_Mesas".EstadoVI[#Mesa].Etapas_Carga_E1 AND NOT "DB900_Estado_Mesas".EstadoVI[#Mesa].Etapas_Carga_E3 AND #Avance_E1_Tx_Ok AND #PosTR_E1 AND "DB902_Estado_ZonaMesa".EstadoMesas[#Mesa].Marcha_CBx AND NOT "DB900_Estado_Mesas".EstadoVI[#Mesa].Error_Mx AND #TP_E3_Dw;
END_REGION

REGION Network 17
   // nieves
   // añadido que no este activa la entrada 1 para darle el permiso a la entrada E2
   RUNG wire#powerrail
      I_Contact( "DB900_Estado_Mesas".EstadoVI[#Mesa].Etapas_Carga_E1 )
      Contact( "DB900_Estado_Mesas".EstadoVI[#Mesa].Etapas_Carga_E3 )
      Contact( #Avance_E3_Tx_Ok )
      Contact( #PosTR_E1 )
      Contact( "DB902_Estado_ZonaMesa".EstadoMesas[#Mesa].Marcha_CBx )
      I_Contact( "DB900_Estado_Mesas".EstadoVI[#Mesa].Error_Mx )
      Contact( #TP_E1_Dw )
      Coil( #PTF_Ent_M3 )
   END_RUNG
   // the same network as SCL:
   #PTF_Ent_M3 := NOT "DB900_Estado_Mesas".EstadoVI[#Mesa].Etapas_Carga_E1 AND "DB900_Estado_Mesas".EstadoVI[#Mesa].Etapas_Carga_E3 AND #Avance_E3_Tx_Ok AND #PosTR_E1 AND "DB902_Estado_ZonaMesa".EstadoMesas[#Mesa].Marcha_CBx AND NOT "DB900_Estado_Mesas".EstadoVI[#Mesa].Error_Mx AND #TP_E1_Dw;
END_REGION

REGION Network 18: Aviso a la Siguiente
   RUNG wire#powerrail
      Contact( "DB900_Estado_Mesas".EstadoVI[#Mesa].Etapa_Cargada )
      wire#w1
      Contact( #PosTR_S2 )
      Contact( "DB902_Estado_ZonaMesa".EstadoMesas[#Mesa].Marcha_CBx )
      I_Contact( "DB900_Estado_Mesas".EstadoVI[#Mesa].Error_Mx )
      Coil( #AVTF_Mx_MSig )
   END_RUNG
   RUNG wire#powerrail
      Contact( "DB900_Estado_Mesas".EstadoVI[#Mesa].Etapas_Descarga_S2 )
   END_RUNG wire#w1
   // the same network as SCL:
   #AVTF_Mx_MSig := ("DB900_Estado_Mesas".EstadoVI[#Mesa].Etapa_Cargada OR "DB900_Estado_Mesas".EstadoVI[#Mesa].Etapas_Descarga_S2) AND #PosTR_S2 AND "DB902_Estado_ZonaMesa".EstadoMesas[#Mesa].Marcha_CBx AND NOT "DB900_Estado_Mesas".EstadoVI[#Mesa].Error_Mx;
END_REGION

REGION Network 19: Salidas Exteriores
   RUNG wire#powerrail
      Contact( "DB900_Estado_Mesas".EstadoVI[#Mesa].Etapa_Vacia )
      I_Contact( #Mem_tmp_Paro )
      Contact( "OFF" )
      wire#w1
      Contact( #PosTR_E1 )
      wire#w4
      Contact( "DB902_Estado_ZonaMesa".EstadoMesas[#Mesa].Marcha_CBx )
      I_Contact( "DB900_Estado_Mesas".EstadoVI[#Mesa].Error_Mx )
      wire#w5
      Contact( #En_Tension )
      Coil( "DB1_SalidasExterioresDeMesa".Mesa[#Mesa].Avanzar_E1E3 )
   END_RUNG
   RUNG wire#powerrail
      Contact( "DB900_Estado_Mesas".EstadoVI[#Mesa].Etapas_Carga_E1 )
      wire#w2
      Contact( #AVTF_Ent_M1 )
      wire#w3
      I_Contact( #OK_Ausencia_Entrada )
   END_RUNG wire#w1
   RUNG wire#w2
      Contact( #pHsMx_E1 )
   END_RUNG wire#w3
   RUNG wire#w2
      Contact( #MemFN_pHsE1 )
   END_RUNG wire#w3
   RUNG wire#w2
      I_Contact( #Mem_tmp_Paro )
   END_RUNG wire#w3
   RUNG wire#w1
      Contact( #TEMP_MA_TR_PosE1E3 )
   END_RUNG wire#w4
   RUNG wire#powerrail
      I_Contact( #Termico_E1_Tx )
      Contact( "DB902_Estado_ZonaMesa".EstadoMesas[#Mesa].Rearme_CBx )
   END_RUNG wire#w5
   // the same network as SCL:
   "DB1_SalidasExterioresDeMesa".Mesa[#Mesa].Avanzar_E1E3 := (((("DB900_Estado_Mesas".EstadoVI[#Mesa].Etapa_Vacia AND NOT #Mem_tmp_Paro AND "OFF") OR ("DB900_Estado_Mesas".EstadoVI[#Mesa].Etapas_Carga_E1 AND (#AVTF_Ent_M1 OR #pHsMx_E1 OR #MemFN_pHsE1 OR NOT #Mem_tmp_Paro) AND NOT #OK_Ausencia_Entrada)) AND (#PosTR_E1 OR #TEMP_MA_TR_PosE1E3) AND "DB902_Estado_ZonaMesa".EstadoMesas[#Mesa].Marcha_CBx AND NOT "DB900_Estado_Mesas".EstadoVI[#Mesa].Error_Mx) OR (NOT #Termico_E1_Tx AND "DB902_Estado_ZonaMesa".EstadoMesas[#Mesa].Rearme_CBx)) AND #En_Tension;
END_REGION

REGION Network 20: ---
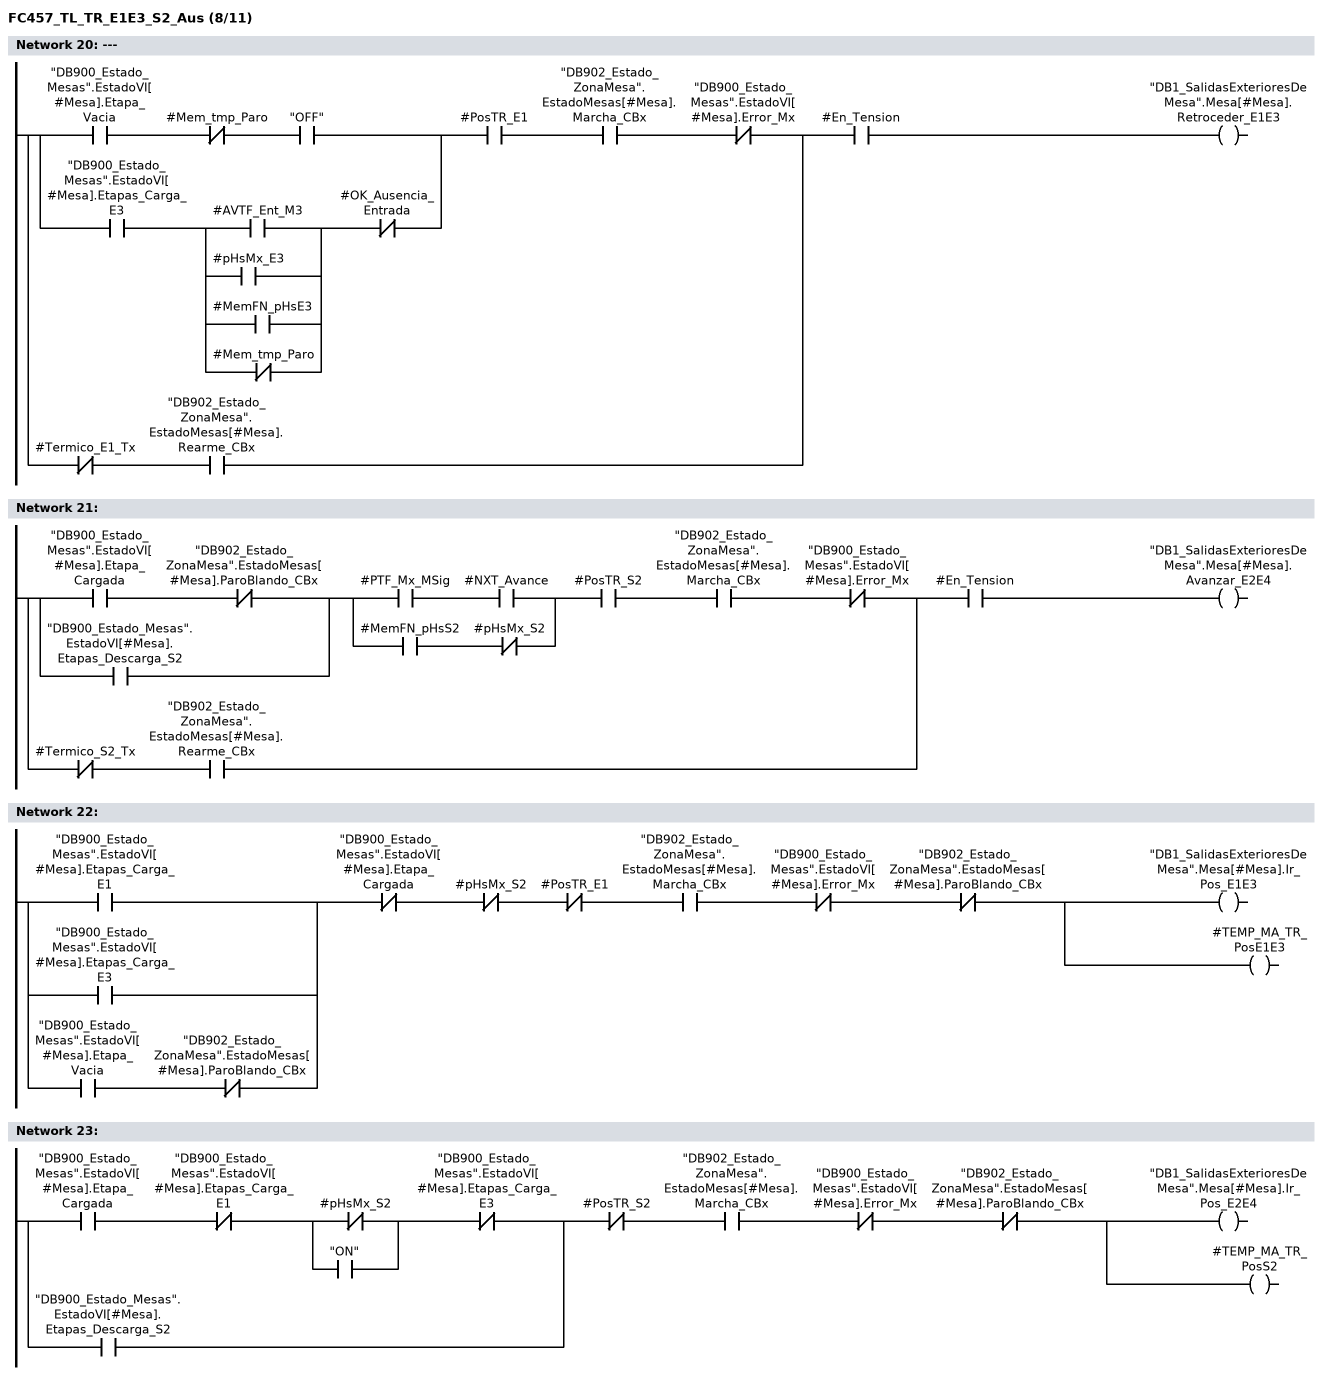
   RUNG wire#powerrail
      Contact( "DB900_Estado_Mesas".EstadoVI[#Mesa].Etapa_Vacia )
      I_Contact( #Mem_tmp_Paro )
      Contact( "OFF" )
      wire#w1
      Contact( #PosTR_E1 )
      Contact( "DB902_Estado_ZonaMesa".EstadoMesas[#Mesa].Marcha_CBx )
      I_Contact( "DB900_Estado_Mesas".EstadoVI[#Mesa].Error_Mx )
      wire#w4
      Contact( #En_Tension )
      Coil( "DB1_SalidasExterioresDeMesa".Mesa[#Mesa].Retroceder_E1E3 )
   END_RUNG
   RUNG wire#powerrail
      Contact( "DB900_Estado_Mesas".EstadoVI[#Mesa].Etapas_Carga_E3 )
      wire#w2
      Contact( #AVTF_Ent_M3 )
      wire#w3
      I_Contact( #OK_Ausencia_Entrada )
   END_RUNG wire#w1
   RUNG wire#w2
      Contact( #pHsMx_E3 )
   END_RUNG wire#w3
   RUNG wire#w2
      Contact( #MemFN_pHsE3 )
   END_RUNG wire#w3
   RUNG wire#w2
      I_Contact( #Mem_tmp_Paro )
   END_RUNG wire#w3
   RUNG wire#powerrail
      I_Contact( #Termico_E1_Tx )
      Contact( "DB902_Estado_ZonaMesa".EstadoMesas[#Mesa].Rearme_CBx )
   END_RUNG wire#w4
   // the same network as SCL:
   "DB1_SalidasExterioresDeMesa".Mesa[#Mesa].Retroceder_E1E3 := (((("DB900_Estado_Mesas".EstadoVI[#Mesa].Etapa_Vacia AND NOT #Mem_tmp_Paro AND "OFF") OR ("DB900_Estado_Mesas".EstadoVI[#Mesa].Etapas_Carga_E3 AND (#AVTF_Ent_M3 OR #pHsMx_E3 OR #MemFN_pHsE3 OR NOT #Mem_tmp_Paro) AND NOT #OK_Ausencia_Entrada)) AND #PosTR_E1 AND "DB902_Estado_ZonaMesa".EstadoMesas[#Mesa].Marcha_CBx AND NOT "DB900_Estado_Mesas".EstadoVI[#Mesa].Error_Mx) OR (NOT #Termico_E1_Tx AND "DB902_Estado_ZonaMesa".EstadoMesas[#Mesa].Rearme_CBx)) AND #En_Tension;
END_REGION

REGION Network 21
   RUNG wire#powerrail
      Contact( "DB900_Estado_Mesas".EstadoVI[#Mesa].Etapa_Cargada )
      I_Contact( "DB902_Estado_ZonaMesa".EstadoMesas[#Mesa].ParoBlando_CBx )
      wire#w1
      Contact( #PTF_Mx_MSig )
      Contact( #NXT_Avance )
      wire#w2
      Contact( #PosTR_S2 )
      Contact( "DB902_Estado_ZonaMesa".EstadoMesas[#Mesa].Marcha_CBx )
      I_Contact( "DB900_Estado_Mesas".EstadoVI[#Mesa].Error_Mx )
      wire#w3
      Contact( #En_Tension )
      Coil( "DB1_SalidasExterioresDeMesa".Mesa[#Mesa].Avanzar_E2E4 )
   END_RUNG
   RUNG wire#powerrail
      Contact( "DB900_Estado_Mesas".EstadoVI[#Mesa].Etapas_Descarga_S2 )
   END_RUNG wire#w1
   RUNG wire#w1
      Contact( #MemFN_pHsS2 )
      I_Contact( #pHsMx_S2 )
   END_RUNG wire#w2
   RUNG wire#powerrail
      I_Contact( #Termico_S2_Tx )
      Contact( "DB902_Estado_ZonaMesa".EstadoMesas[#Mesa].Rearme_CBx )
   END_RUNG wire#w3
   // the same network as SCL:
   "DB1_SalidasExterioresDeMesa".Mesa[#Mesa].Avanzar_E2E4 := (((("DB900_Estado_Mesas".EstadoVI[#Mesa].Etapa_Cargada AND NOT "DB902_Estado_ZonaMesa".EstadoMesas[#Mesa].ParoBlando_CBx) OR "DB900_Estado_Mesas".EstadoVI[#Mesa].Etapas_Descarga_S2) AND ((#PTF_Mx_MSig AND #NXT_Avance) OR (#MemFN_pHsS2 AND NOT #pHsMx_S2)) AND #PosTR_S2 AND "DB902_Estado_ZonaMesa".EstadoMesas[#Mesa].Marcha_CBx AND NOT "DB900_Estado_Mesas".EstadoVI[#Mesa].Error_Mx) OR (NOT #Termico_S2_Tx AND "DB902_Estado_ZonaMesa".EstadoMesas[#Mesa].Rearme_CBx)) AND #En_Tension;
END_REGION

REGION Network 22
   RUNG wire#powerrail
      Contact( "DB900_Estado_Mesas".EstadoVI[#Mesa].Etapas_Carga_E1 )
      wire#w1
      I_Contact( "DB900_Estado_Mesas".EstadoVI[#Mesa].Etapa_Cargada )
      I_Contact( #pHsMx_S2 )
      I_Contact( #PosTR_E1 )
      Contact( "DB902_Estado_ZonaMesa".EstadoMesas[#Mesa].Marcha_CBx )
      I_Contact( "DB900_Estado_Mesas".EstadoVI[#Mesa].Error_Mx )
      I_Contact( "DB902_Estado_ZonaMesa".EstadoMesas[#Mesa].ParoBlando_CBx )
      wire#w2
      Coil( "DB1_SalidasExterioresDeMesa".Mesa[#Mesa].Ir_Pos_E1E3 )
   END_RUNG
   RUNG wire#powerrail
      Contact( "DB900_Estado_Mesas".EstadoVI[#Mesa].Etapas_Carga_E3 )
   END_RUNG wire#w1
   RUNG wire#powerrail
      Contact( "DB900_Estado_Mesas".EstadoVI[#Mesa].Etapa_Vacia )
      I_Contact( "DB902_Estado_ZonaMesa".EstadoMesas[#Mesa].ParoBlando_CBx )
   END_RUNG wire#w1
   RUNG wire#w2
      Coil( #TEMP_MA_TR_PosE1E3 )
   END_RUNG
   // the same network as SCL:
   #_w1 := ("DB900_Estado_Mesas".EstadoVI[#Mesa].Etapas_Carga_E1 OR "DB900_Estado_Mesas".EstadoVI[#Mesa].Etapas_Carga_E3 OR ("DB900_Estado_Mesas".EstadoVI[#Mesa].Etapa_Vacia AND NOT "DB902_Estado_ZonaMesa".EstadoMesas[#Mesa].ParoBlando_CBx)) AND NOT "DB900_Estado_Mesas".EstadoVI[#Mesa].Etapa_Cargada AND NOT #pHsMx_S2 AND NOT #PosTR_E1 AND "DB902_Estado_ZonaMesa".EstadoMesas[#Mesa].Marcha_CBx AND NOT "DB900_Estado_Mesas".EstadoVI[#Mesa].Error_Mx AND NOT "DB902_Estado_ZonaMesa".EstadoMesas[#Mesa].ParoBlando_CBx;
   "DB1_SalidasExterioresDeMesa".Mesa[#Mesa].Ir_Pos_E1E3 := ("DB900_Estado_Mesas".EstadoVI[#Mesa].Etapas_Carga_E1 OR "DB900_Estado_Mesas".EstadoVI[#Mesa].Etapas_Carga_E3 OR ("DB900_Estado_Mesas".EstadoVI[#Mesa].Etapa_Vacia AND NOT "DB902_Estado_ZonaMesa".EstadoMesas[#Mesa].ParoBlando_CBx)) AND NOT "DB900_Estado_Mesas".EstadoVI[#Mesa].Etapa_Cargada AND NOT #pHsMx_S2 AND NOT #PosTR_E1 AND "DB902_Estado_ZonaMesa".EstadoMesas[#Mesa].Marcha_CBx AND NOT "DB900_Estado_Mesas".EstadoVI[#Mesa].Error_Mx AND NOT "DB902_Estado_ZonaMesa".EstadoMesas[#Mesa].ParoBlando_CBx;
   #TEMP_MA_TR_PosE1E3 := #_w1;
END_REGION

REGION Network 23
   RUNG wire#powerrail
      Contact( "DB900_Estado_Mesas".EstadoVI[#Mesa].Etapa_Cargada )
      I_Contact( "DB900_Estado_Mesas".EstadoVI[#Mesa].Etapas_Carga_E1 )
      wire#w1
      I_Contact( #pHsMx_S2 )
      wire#w2
      I_Contact( "DB900_Estado_Mesas".EstadoVI[#Mesa].Etapas_Carga_E3 )
      wire#w3
      I_Contact( #PosTR_S2 )
      Contact( "DB902_Estado_ZonaMesa".EstadoMesas[#Mesa].Marcha_CBx )
      I_Contact( "DB900_Estado_Mesas".EstadoVI[#Mesa].Error_Mx )
      I_Contact( "DB902_Estado_ZonaMesa".EstadoMesas[#Mesa].ParoBlando_CBx )
      wire#w4
      Coil( "DB1_SalidasExterioresDeMesa".Mesa[#Mesa].Ir_Pos_E2E4 )
   END_RUNG
   RUNG wire#w1
      Contact( "ON" )
   END_RUNG wire#w2
   RUNG wire#powerrail
      Contact( "DB900_Estado_Mesas".EstadoVI[#Mesa].Etapas_Descarga_S2 )
   END_RUNG wire#w3
   RUNG wire#w4
      Coil( #TEMP_MA_TR_PosS2 )
   END_RUNG
   // the same network as SCL:
   #_w1 := (("DB900_Estado_Mesas".EstadoVI[#Mesa].Etapa_Cargada AND NOT "DB900_Estado_Mesas".EstadoVI[#Mesa].Etapas_Carga_E1 AND (NOT #pHsMx_S2 OR "ON") AND NOT "DB900_Estado_Mesas".EstadoVI[#Mesa].Etapas_Carga_E3) OR "DB900_Estado_Mesas".EstadoVI[#Mesa].Etapas_Descarga_S2) AND NOT #PosTR_S2 AND "DB902_Estado_ZonaMesa".EstadoMesas[#Mesa].Marcha_CBx AND NOT "DB900_Estado_Mesas".EstadoVI[#Mesa].Error_Mx AND NOT "DB902_Estado_ZonaMesa".EstadoMesas[#Mesa].ParoBlando_CBx;
   "DB1_SalidasExterioresDeMesa".Mesa[#Mesa].Ir_Pos_E2E4 := (("DB900_Estado_Mesas".EstadoVI[#Mesa].Etapa_Cargada AND NOT "DB900_Estado_Mesas".EstadoVI[#Mesa].Etapas_Carga_E1 AND (NOT #pHsMx_S2 OR "ON") AND NOT "DB900_Estado_Mesas".EstadoVI[#Mesa].Etapas_Carga_E3) OR "DB900_Estado_Mesas".EstadoVI[#Mesa].Etapas_Descarga_S2) AND NOT #PosTR_S2 AND "DB902_Estado_ZonaMesa".EstadoMesas[#Mesa].Marcha_CBx AND NOT "DB900_Estado_Mesas".EstadoVI[#Mesa].Error_Mx AND NOT "DB902_Estado_ZonaMesa".EstadoMesas[#Mesa].ParoBlando_CBx;
   #TEMP_MA_TR_PosS2 := #_w1;
END_REGION

REGION Network 24: Subida de topes
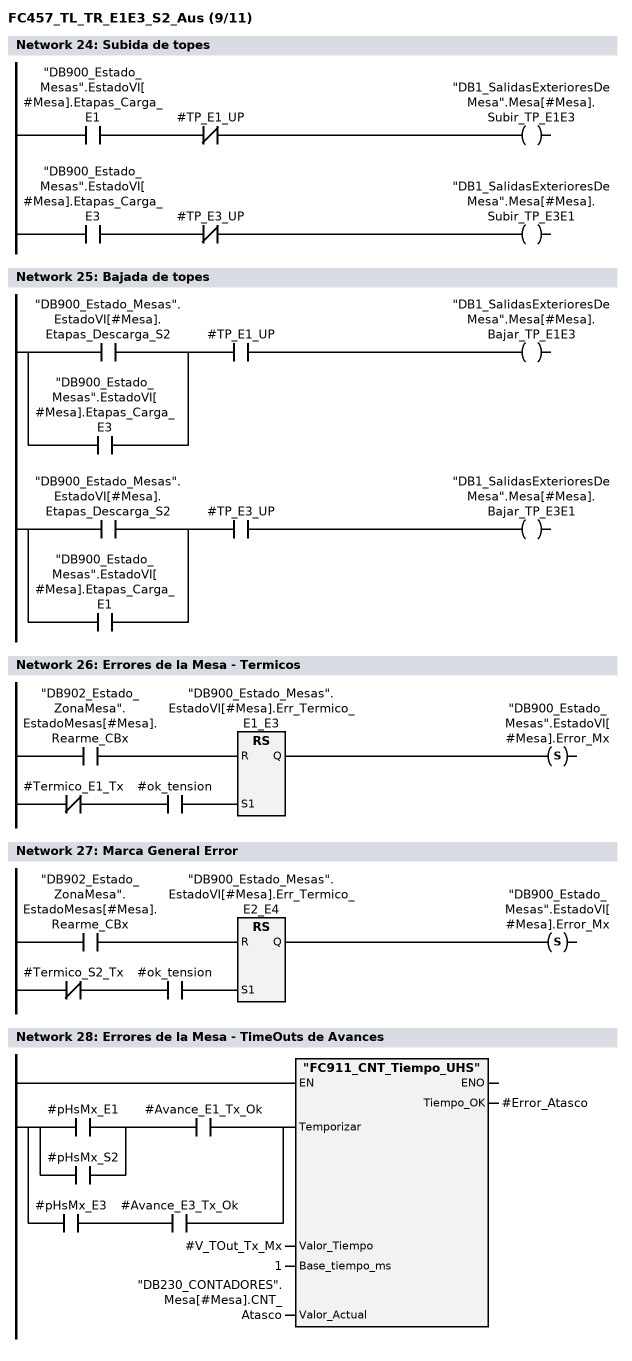
   RUNG wire#powerrail
      Contact( "DB900_Estado_Mesas".EstadoVI[#Mesa].Etapas_Carga_E1 )
      I_Contact( #TP_E1_UP )
      Coil( "DB1_SalidasExterioresDeMesa".Mesa[#Mesa].Subir_TP_E1E3 )
   END_RUNG
   RUNG wire#powerrail
      Contact( "DB900_Estado_Mesas".EstadoVI[#Mesa].Etapas_Carga_E3 )
      I_Contact( #TP_E3_UP )
      Coil( "DB1_SalidasExterioresDeMesa".Mesa[#Mesa].Subir_TP_E3E1 )
   END_RUNG
   // the same network as SCL:
   "DB1_SalidasExterioresDeMesa".Mesa[#Mesa].Subir_TP_E1E3 := "DB900_Estado_Mesas".EstadoVI[#Mesa].Etapas_Carga_E1 AND NOT #TP_E1_UP;
   "DB1_SalidasExterioresDeMesa".Mesa[#Mesa].Subir_TP_E3E1 := "DB900_Estado_Mesas".EstadoVI[#Mesa].Etapas_Carga_E3 AND NOT #TP_E3_UP;
END_REGION

REGION Network 25: Bajada de topes
   RUNG wire#powerrail
      Contact( "DB900_Estado_Mesas".EstadoVI[#Mesa].Etapas_Descarga_S2 )
      wire#w1
      Contact( #TP_E1_UP )
      Coil( "DB1_SalidasExterioresDeMesa".Mesa[#Mesa].Bajar_TP_E1E3 )
   END_RUNG
   RUNG wire#powerrail
      Contact( "DB900_Estado_Mesas".EstadoVI[#Mesa].Etapas_Carga_E3 )
   END_RUNG wire#w1
   RUNG wire#powerrail
      Contact( "DB900_Estado_Mesas".EstadoVI[#Mesa].Etapas_Descarga_S2 )
      wire#w2
      Contact( #TP_E3_UP )
      Coil( "DB1_SalidasExterioresDeMesa".Mesa[#Mesa].Bajar_TP_E3E1 )
   END_RUNG
   RUNG wire#powerrail
      Contact( "DB900_Estado_Mesas".EstadoVI[#Mesa].Etapas_Carga_E1 )
   END_RUNG wire#w2
   // the same network as SCL:
   "DB1_SalidasExterioresDeMesa".Mesa[#Mesa].Bajar_TP_E1E3 := ("DB900_Estado_Mesas".EstadoVI[#Mesa].Etapas_Descarga_S2 OR "DB900_Estado_Mesas".EstadoVI[#Mesa].Etapas_Carga_E3) AND #TP_E1_UP;
   "DB1_SalidasExterioresDeMesa".Mesa[#Mesa].Bajar_TP_E3E1 := ("DB900_Estado_Mesas".EstadoVI[#Mesa].Etapas_Descarga_S2 OR "DB900_Estado_Mesas".EstadoVI[#Mesa].Etapas_Carga_E1) AND #TP_E3_UP;
END_REGION

REGION Network 26: Errores de la Mesa - Termicos
   RUNG wire#powerrail
      Contact( "DB902_Estado_ZonaMesa".EstadoMesas[#Mesa].Rearme_CBx )
      S_RS(operand := "DB900_Estado_Mesas".EstadoVI[#Mesa].Err_Termico_E1_E3, s1 := wire#w1)
      S_Coil( "DB900_Estado_Mesas".EstadoVI[#Mesa].Error_Mx )
   END_RUNG
   RUNG wire#powerrail
      I_Contact( #Termico_E1_Tx )
      Contact( #ok_tension )
   END_RUNG wire#w1
   // the same network as SCL:
   IF "DB902_Estado_ZonaMesa".EstadoMesas[#Mesa].Rearme_CBx THEN
       "DB900_Estado_Mesas".EstadoVI[#Mesa].Err_Termico_E1_E3 := FALSE;   // RS flip-flop
   END_IF;
   IF NOT #Termico_E1_Tx AND #ok_tension THEN
       "DB900_Estado_Mesas".EstadoVI[#Mesa].Err_Termico_E1_E3 := TRUE;
   END_IF;
   IF "DB900_Estado_Mesas".EstadoVI[#Mesa].Err_Termico_E1_E3 THEN
       "DB900_Estado_Mesas".EstadoVI[#Mesa].Error_Mx := TRUE;
   END_IF;
END_REGION

REGION Network 27: Marca General Error
   RUNG wire#powerrail
      Contact( "DB902_Estado_ZonaMesa".EstadoMesas[#Mesa].Rearme_CBx )
      S_RS(operand := "DB900_Estado_Mesas".EstadoVI[#Mesa].Err_Termico_E2_E4, s1 := wire#w1)
      S_Coil( "DB900_Estado_Mesas".EstadoVI[#Mesa].Error_Mx )
   END_RUNG
   RUNG wire#powerrail
      I_Contact( #Termico_S2_Tx )
      Contact( #ok_tension )
   END_RUNG wire#w1
   // the same network as SCL:
   IF "DB902_Estado_ZonaMesa".EstadoMesas[#Mesa].Rearme_CBx THEN
       "DB900_Estado_Mesas".EstadoVI[#Mesa].Err_Termico_E2_E4 := FALSE;   // RS flip-flop
   END_IF;
   IF NOT #Termico_S2_Tx AND #ok_tension THEN
       "DB900_Estado_Mesas".EstadoVI[#Mesa].Err_Termico_E2_E4 := TRUE;
   END_IF;
   IF "DB900_Estado_Mesas".EstadoVI[#Mesa].Err_Termico_E2_E4 THEN
       "DB900_Estado_Mesas".EstadoVI[#Mesa].Error_Mx := TRUE;
   END_IF;
END_REGION

REGION Network 28: Errores de la Mesa - TimeOuts de Avances
   RUNG wire#powerrail
      "FC911_CNT_Tiempo_UHS"(Temporizar := wire#w2, Valor_Tiempo := #V_TOut_Tx_Mx, Base_tiempo_ms := 1, Valor_Actual := "DB230_CONTADORES".Mesa[#Mesa].CNT_Atasco, Tiempo_OK => #Error_Atasco)
   END_RUNG
   RUNG wire#powerrail
      Contact( #pHsMx_E1 )
      wire#w1
      Contact( #Avance_E1_Tx_Ok )
   END_RUNG wire#w2
   RUNG wire#powerrail
      Contact( #pHsMx_S2 )
   END_RUNG wire#w1
   RUNG wire#powerrail
      Contact( #pHsMx_E3 )
      Contact( #Avance_E3_Tx_Ok )
   END_RUNG wire#w2
   // the same network as SCL:
   "FC911_CNT_Tiempo_UHS"(Temporizar := ((#pHsMx_E1 OR #pHsMx_S2) AND #Avance_E1_Tx_Ok) OR (#pHsMx_E3 AND #Avance_E3_Tx_Ok),
                          Valor_Tiempo := #V_TOut_Tx_Mx,
                          Base_tiempo_ms := 1,
                          Valor_Actual := "DB230_CONTADORES".Mesa[#Mesa].CNT_Atasco,
                          Tiempo_OK => #Error_Atasco);
END_REGION

REGION Network 29
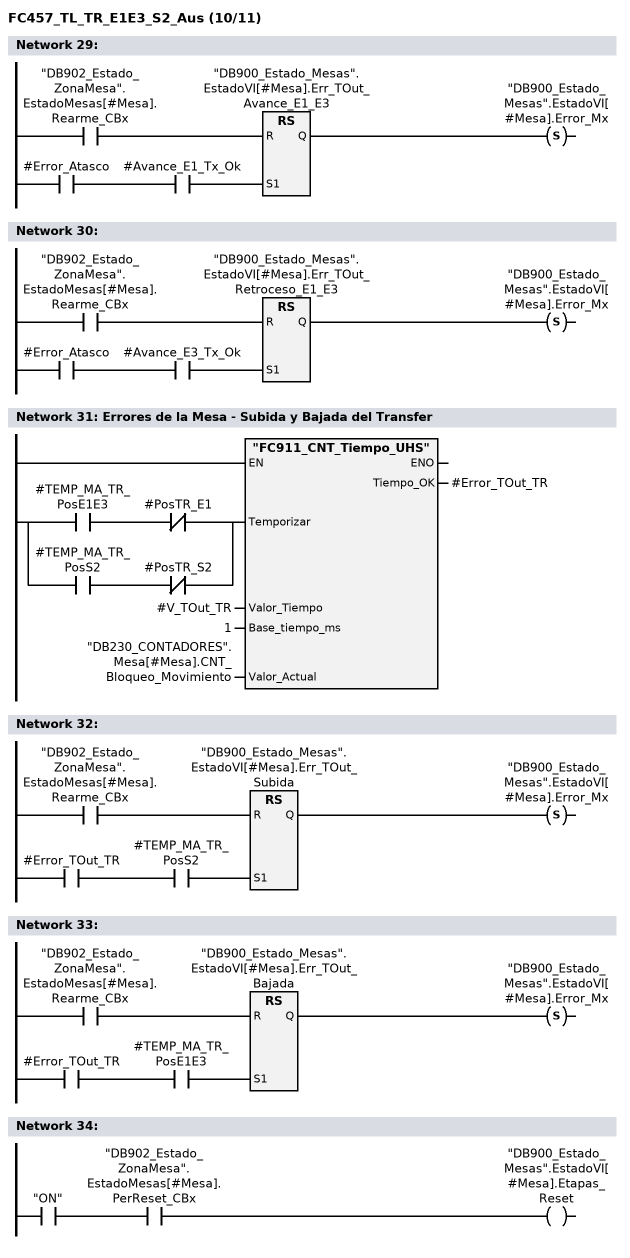
   RUNG wire#powerrail
      Contact( "DB902_Estado_ZonaMesa".EstadoMesas[#Mesa].Rearme_CBx )
      S_RS(operand := "DB900_Estado_Mesas".EstadoVI[#Mesa].Err_TOut_Avance_E1_E3, s1 := wire#w1)
      S_Coil( "DB900_Estado_Mesas".EstadoVI[#Mesa].Error_Mx )
   END_RUNG
   RUNG wire#powerrail
      Contact( #Error_Atasco )
      Contact( #Avance_E1_Tx_Ok )
   END_RUNG wire#w1
   // the same network as SCL:
   IF "DB902_Estado_ZonaMesa".EstadoMesas[#Mesa].Rearme_CBx THEN
       "DB900_Estado_Mesas".EstadoVI[#Mesa].Err_TOut_Avance_E1_E3 := FALSE;   // RS flip-flop
   END_IF;
   IF #Error_Atasco AND #Avance_E1_Tx_Ok THEN
       "DB900_Estado_Mesas".EstadoVI[#Mesa].Err_TOut_Avance_E1_E3 := TRUE;
   END_IF;
   IF "DB900_Estado_Mesas".EstadoVI[#Mesa].Err_TOut_Avance_E1_E3 THEN
       "DB900_Estado_Mesas".EstadoVI[#Mesa].Error_Mx := TRUE;
   END_IF;
END_REGION

REGION Network 30
   RUNG wire#powerrail
      Contact( "DB902_Estado_ZonaMesa".EstadoMesas[#Mesa].Rearme_CBx )
      S_RS(operand := "DB900_Estado_Mesas".EstadoVI[#Mesa].Err_TOut_Retroceso_E1_E3, s1 := wire#w1)
      S_Coil( "DB900_Estado_Mesas".EstadoVI[#Mesa].Error_Mx )
   END_RUNG
   RUNG wire#powerrail
      Contact( #Error_Atasco )
      Contact( #Avance_E3_Tx_Ok )
   END_RUNG wire#w1
   // the same network as SCL:
   IF "DB902_Estado_ZonaMesa".EstadoMesas[#Mesa].Rearme_CBx THEN
       "DB900_Estado_Mesas".EstadoVI[#Mesa].Err_TOut_Retroceso_E1_E3 := FALSE;   // RS flip-flop
   END_IF;
   IF #Error_Atasco AND #Avance_E3_Tx_Ok THEN
       "DB900_Estado_Mesas".EstadoVI[#Mesa].Err_TOut_Retroceso_E1_E3 := TRUE;
   END_IF;
   IF "DB900_Estado_Mesas".EstadoVI[#Mesa].Err_TOut_Retroceso_E1_E3 THEN
       "DB900_Estado_Mesas".EstadoVI[#Mesa].Error_Mx := TRUE;
   END_IF;
END_REGION

REGION Network 31: Errores de la Mesa - Subida y Bajada del Transfer
   RUNG wire#powerrail
      "FC911_CNT_Tiempo_UHS"(Temporizar := wire#w1, Valor_Tiempo := #V_TOut_TR, Base_tiempo_ms := 1, Valor_Actual := "DB230_CONTADORES".Mesa[#Mesa].CNT_Bloqueo_Movimiento, Tiempo_OK => #Error_TOut_TR)
   END_RUNG
   RUNG wire#powerrail
      Contact( #TEMP_MA_TR_PosE1E3 )
      I_Contact( #PosTR_E1 )
   END_RUNG wire#w1
   RUNG wire#powerrail
      Contact( #TEMP_MA_TR_PosS2 )
      I_Contact( #PosTR_S2 )
   END_RUNG wire#w1
   // the same network as SCL:
   "FC911_CNT_Tiempo_UHS"(Temporizar := (#TEMP_MA_TR_PosE1E3 AND NOT #PosTR_E1) OR (#TEMP_MA_TR_PosS2 AND NOT #PosTR_S2),
                          Valor_Tiempo := #V_TOut_TR,
                          Base_tiempo_ms := 1,
                          Valor_Actual := "DB230_CONTADORES".Mesa[#Mesa].CNT_Bloqueo_Movimiento,
                          Tiempo_OK => #Error_TOut_TR);
END_REGION

REGION Network 32
   RUNG wire#powerrail
      Contact( "DB902_Estado_ZonaMesa".EstadoMesas[#Mesa].Rearme_CBx )
      S_RS(operand := "DB900_Estado_Mesas".EstadoVI[#Mesa].Err_TOut_Subida, s1 := wire#w1)
      S_Coil( "DB900_Estado_Mesas".EstadoVI[#Mesa].Error_Mx )
   END_RUNG
   RUNG wire#powerrail
      Contact( #Error_TOut_TR )
      Contact( #TEMP_MA_TR_PosS2 )
   END_RUNG wire#w1
   // the same network as SCL:
   IF "DB902_Estado_ZonaMesa".EstadoMesas[#Mesa].Rearme_CBx THEN
       "DB900_Estado_Mesas".EstadoVI[#Mesa].Err_TOut_Subida := FALSE;   // RS flip-flop
   END_IF;
   IF #Error_TOut_TR AND #TEMP_MA_TR_PosS2 THEN
       "DB900_Estado_Mesas".EstadoVI[#Mesa].Err_TOut_Subida := TRUE;
   END_IF;
   IF "DB900_Estado_Mesas".EstadoVI[#Mesa].Err_TOut_Subida THEN
       "DB900_Estado_Mesas".EstadoVI[#Mesa].Error_Mx := TRUE;
   END_IF;
END_REGION

REGION Network 33
   RUNG wire#powerrail
      Contact( "DB902_Estado_ZonaMesa".EstadoMesas[#Mesa].Rearme_CBx )
      S_RS(operand := "DB900_Estado_Mesas".EstadoVI[#Mesa].Err_TOut_Bajada, s1 := wire#w1)
      S_Coil( "DB900_Estado_Mesas".EstadoVI[#Mesa].Error_Mx )
   END_RUNG
   RUNG wire#powerrail
      Contact( #Error_TOut_TR )
      Contact( #TEMP_MA_TR_PosE1E3 )
   END_RUNG wire#w1
   // the same network as SCL:
   IF "DB902_Estado_ZonaMesa".EstadoMesas[#Mesa].Rearme_CBx THEN
       "DB900_Estado_Mesas".EstadoVI[#Mesa].Err_TOut_Bajada := FALSE;   // RS flip-flop
   END_IF;
   IF #Error_TOut_TR AND #TEMP_MA_TR_PosE1E3 THEN
       "DB900_Estado_Mesas".EstadoVI[#Mesa].Err_TOut_Bajada := TRUE;
   END_IF;
   IF "DB900_Estado_Mesas".EstadoVI[#Mesa].Err_TOut_Bajada THEN
       "DB900_Estado_Mesas".EstadoVI[#Mesa].Error_Mx := TRUE;
   END_IF;
END_REGION

REGION Network 34
   RUNG wire#powerrail
      Contact( "ON" )
      Contact( "DB902_Estado_ZonaMesa".EstadoMesas[#Mesa].PerReset_CBx )
      Coil( "DB900_Estado_Mesas".EstadoVI[#Mesa].Etapas_Reset )
   END_RUNG
   // the same network as SCL:
   "DB900_Estado_Mesas".EstadoVI[#Mesa].Etapas_Reset := "ON" AND "DB902_Estado_ZonaMesa".EstadoMesas[#Mesa].PerReset_CBx;
END_REGION

REGION Network 35: Entradas Mesas
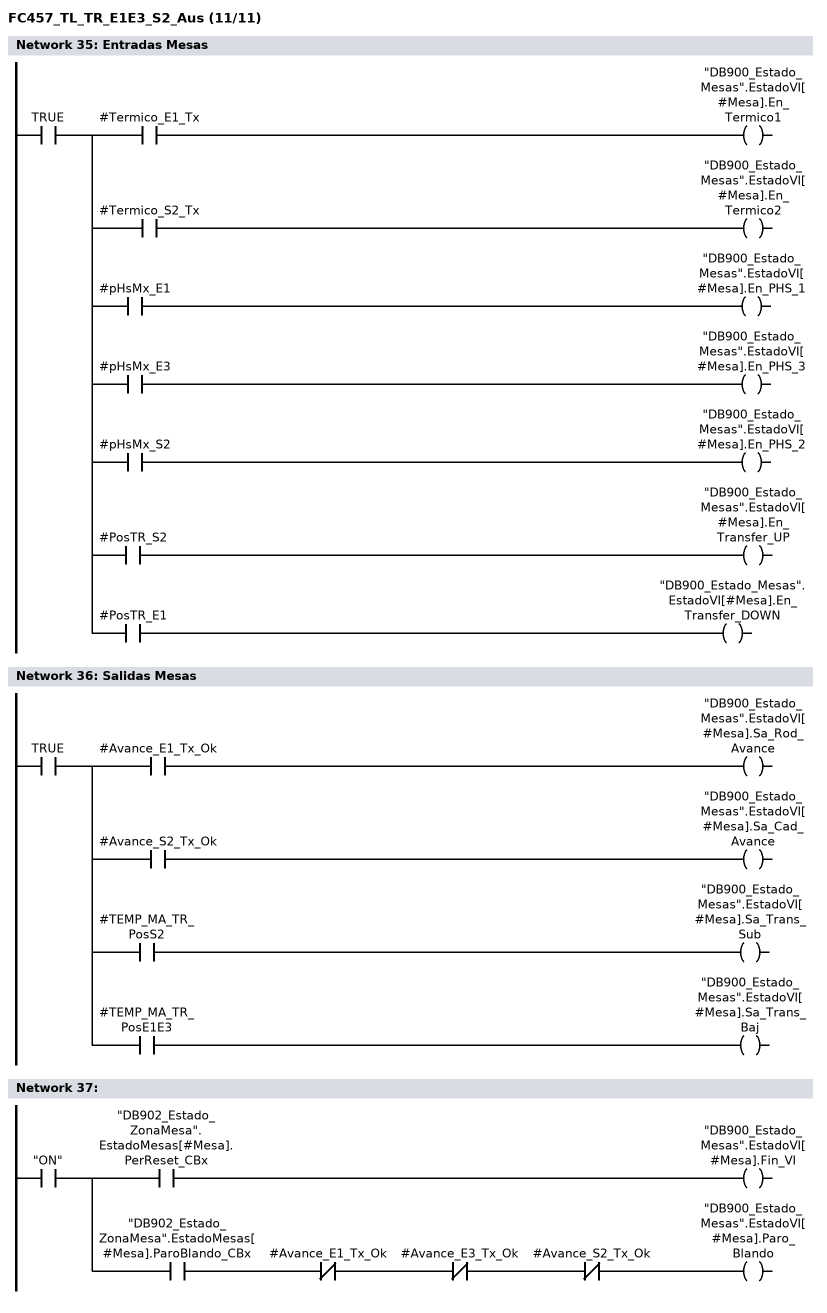
   RUNG wire#powerrail
      Contact( TRUE )
      wire#w1
      Contact( #Termico_E1_Tx )
      Coil( "DB900_Estado_Mesas".EstadoVI[#Mesa].En_Termico1 )
   END_RUNG
   RUNG wire#w1
      Contact( #Termico_S2_Tx )
      Coil( "DB900_Estado_Mesas".EstadoVI[#Mesa].En_Termico2 )
   END_RUNG
   RUNG wire#w1
      Contact( #pHsMx_E1 )
      Coil( "DB900_Estado_Mesas".EstadoVI[#Mesa].En_PHS_1 )
   END_RUNG
   RUNG wire#w1
      Contact( #pHsMx_E3 )
      Coil( "DB900_Estado_Mesas".EstadoVI[#Mesa].En_PHS_3 )
   END_RUNG
   RUNG wire#w1
      Contact( #pHsMx_S2 )
      Coil( "DB900_Estado_Mesas".EstadoVI[#Mesa].En_PHS_2 )
   END_RUNG
   RUNG wire#w1
      Contact( #PosTR_S2 )
      Coil( "DB900_Estado_Mesas".EstadoVI[#Mesa].En_Transfer_UP )
   END_RUNG
   RUNG wire#w1
      Contact( #PosTR_E1 )
      Coil( "DB900_Estado_Mesas".EstadoVI[#Mesa].En_Transfer_DOWN )
   END_RUNG
   // the same network as SCL:
   "DB900_Estado_Mesas".EstadoVI[#Mesa].En_Termico1 := TRUE AND #Termico_E1_Tx;
   "DB900_Estado_Mesas".EstadoVI[#Mesa].En_Termico2 := TRUE AND #Termico_S2_Tx;
   "DB900_Estado_Mesas".EstadoVI[#Mesa].En_PHS_1 := TRUE AND #pHsMx_E1;
   "DB900_Estado_Mesas".EstadoVI[#Mesa].En_PHS_3 := TRUE AND #pHsMx_E3;
   "DB900_Estado_Mesas".EstadoVI[#Mesa].En_PHS_2 := TRUE AND #pHsMx_S2;
   "DB900_Estado_Mesas".EstadoVI[#Mesa].En_Transfer_UP := TRUE AND #PosTR_S2;
   "DB900_Estado_Mesas".EstadoVI[#Mesa].En_Transfer_DOWN := TRUE AND #PosTR_E1;
END_REGION

REGION Network 36: Salidas Mesas
   RUNG wire#powerrail
      Contact( TRUE )
      wire#w1
      Contact( #Avance_E1_Tx_Ok )
      Coil( "DB900_Estado_Mesas".EstadoVI[#Mesa].Sa_Rod_Avance )
   END_RUNG
   RUNG wire#w1
      Contact( #Avance_S2_Tx_Ok )
      Coil( "DB900_Estado_Mesas".EstadoVI[#Mesa].Sa_Cad_Avance )
   END_RUNG
   RUNG wire#w1
      Contact( #TEMP_MA_TR_PosS2 )
      Coil( "DB900_Estado_Mesas".EstadoVI[#Mesa].Sa_Trans_Sub )
   END_RUNG
   RUNG wire#w1
      Contact( #TEMP_MA_TR_PosE1E3 )
      Coil( "DB900_Estado_Mesas".EstadoVI[#Mesa].Sa_Trans_Baj )
   END_RUNG
   // the same network as SCL:
   "DB900_Estado_Mesas".EstadoVI[#Mesa].Sa_Rod_Avance := TRUE AND #Avance_E1_Tx_Ok;
   "DB900_Estado_Mesas".EstadoVI[#Mesa].Sa_Cad_Avance := TRUE AND #Avance_S2_Tx_Ok;
   "DB900_Estado_Mesas".EstadoVI[#Mesa].Sa_Trans_Sub := TRUE AND #TEMP_MA_TR_PosS2;
   "DB900_Estado_Mesas".EstadoVI[#Mesa].Sa_Trans_Baj := TRUE AND #TEMP_MA_TR_PosE1E3;
END_REGION

REGION Network 37
   RUNG wire#powerrail
      Contact( "ON" )
      wire#w1
      Contact( "DB902_Estado_ZonaMesa".EstadoMesas[#Mesa].PerReset_CBx )
      Coil( "DB900_Estado_Mesas".EstadoVI[#Mesa].Fin_VI )
   END_RUNG
   RUNG wire#w1
      Contact( "DB902_Estado_ZonaMesa".EstadoMesas[#Mesa].ParoBlando_CBx )
      I_Contact( #Avance_E1_Tx_Ok )
      I_Contact( #Avance_E3_Tx_Ok )
      I_Contact( #Avance_S2_Tx_Ok )
      Coil( "DB900_Estado_Mesas".EstadoVI[#Mesa].Paro_Blando )
   END_RUNG
   // the same network as SCL:
   "DB900_Estado_Mesas".EstadoVI[#Mesa].Fin_VI := "ON" AND "DB902_Estado_ZonaMesa".EstadoMesas[#Mesa].PerReset_CBx;
   "DB900_Estado_Mesas".EstadoVI[#Mesa].Paro_Blando := "ON" AND "DB902_Estado_ZonaMesa".EstadoMesas[#Mesa].ParoBlando_CBx AND NOT #Avance_E1_Tx_Ok AND NOT #Avance_E3_Tx_Ok AND NOT #Avance_S2_Tx_Ok;
END_REGION
END_FUNCTION
